# B&R Automation Studio project PLC code - cp (part 11)

#### InksCtrl.var
```iecst
VAR
	uiPosTachoCounterPrev : UINT;
	uiNegTachoCounterPrev : UINT;
	uiMode1Cycles : UINT;
	uiMode3Cycles : UINT;
	uiMode4Cycles : UINT;
	uiMode5Cycles : UINT;
	uiMode6Cycles : UINT;
	uiMode9Cycles : UINT;
	uiMode10Cycles : UINT;
	uiMode13Cycles : UINT;
	TON_AlrVacuum1 : TON;
	tonInkLevelBelowMinimum : TON;
	tonInkLevelBelowCloseMinimum : TON;
	TON_StabSolPid2Pos : TON; (*Vars Pressure Control*)
	TON_ChangeSPstarting : TON; (*It is a delay to recovery original set point after differential pressures*)
	TON_CloseSole : TON;
	tonInkLevelBelowMaximum : TON;
	TON_AlrTempGauge : TON;
	TON_HeaterStarts : TON;
	TON_AlrVacuum2 : TON;
	TON_OnReverseCappedCycle : TON; (*timer 30 min. It is cylce of reverse cleaning in Idle*)
	tonInkLevelAboveMaximum : TON;
	TON_DelayVacuum2Gauge : TON;
	tonInkLevelAboveMinimum : TON;
	TON_Stab2 : TON;
	TON_Stab1 : TON;
	TON_StabSolPid2Neg : TON;
	TON_TimeAfterCloseReliefValve : TON;
	TON_ChangeSPInDelta : TON; (*It is a delay to recovery original set point after differential pressures*) (*stChangeSPstarted : TON; *) (*It is a delay to recovery original set point after differential pressures*)
	TON_DelayVacuum1Gauge : TON;
	TON_ExecutionDelay : TON; (*Delay to activate the PID's in order to be sure to have proper configuration*)
	TON_AlrVacuumDiff2 : TON;
	TON_StabPsuOk : TON;
	TON_AlrNegDiff : TON;
	TON_StabSolPid1Neg : TON;
	TON_ChangeReverse : TON;
	TON_AlrDCDiff : TON;
	TON_AlrCriticalMeniscus2 : TON;
	TON_AlrNotDifTemp : TON;
	TON_TimeAlrDCStarting : TON;
	TON_AlrPosDiff : TON;
	TON_AlrIncoherTempHeat : TON;
	TON_AlrDifTemp : TON;
	TON_AlrVacuumDiff : TON;
	TON_StabSolPid1Pos : TON;
	TON_ChangeFillingControl : TON;
	TON_Reset : TON;
	TON_OnStateReverseFlow : TON; (*More time than 30 secs because It is coming back on reverse state *)
	TON_OnReverseCappedFinished : TON; (*timer 60 secs. It is time reverse cleaning in Idle*)
	TON_TimeExecutingReverseMan : TON;
	TON_Stopped : TON;
	TON_PressureReservoirStable : TON;
	TOF_IgnoreAlarmsCleaning : TOF;
	tonDrip : TON;
	parBar : REFERENCE TO stInksBarParams;
	inks : REFERENCE TO stInks;
	r_start_inks : R_TRIG;
	rSlopePumpNeg : REAL;
	rSPfillingPump : REAL; (*Value directly from Sw*)
	rPressureCollectorPos1 : REAL; (*REVISAR, sale un mensaje al traducir*)
	rSlopePumpPos : REAL;
	rSpeedNegCalc : REAL;
	rPressureCollectorPos2 : REAL; (*REVISAR, sale un mensaje al traducir*)
	rPressurePos : REAL;
	rPressureMen : REAL;
	rSP_NegPrimStabilizing : REAL;
	rSP_PosPrimStabilizing : REAL;
	rTankLevelmm : REAL;
	rSetPointFillingPump : REAL; (*Vars Temp Control*)
	rOrderBNegative : REAL;
	rVoltagePosPump : REAL;
	rOrderBPositiveStart : REAL;
	rOrderBPositive : REAL;
	rSP_Meniscus_PID : REAL;
	rMeniscusSp : REAL; (*Value directly from Sw*)
	rMeniscusPV : REAL;
	rVacuum2B : REAL;
	rSPTempTank : REAL;
	rHighPumpLimitNeg : REAL;
	rHighPumpLimitPos : REAL;
	rVoltageNegPump : REAL;
	rInputFilterVacuum2 : REAL;
	rLowPumpLimitNeg : REAL;
	parPidPos : REAL;
	parPidPosCopy : REAL;
	rInputFilterVacuum1 : REAL;
	parPidMeniscus : REAL;
	parPidMeniscusCopy : REAL;
	rSpeedPosCalc : REAL;
	parPidTemp : REAL;
	parPidTempCopy : REAL;
	rSPtemp : REAL; (*Temperature SetPoint*)
	rDutyCyclePreTune : REAL;
	rDutyCycleTempAux : REAL;
	rTankLevelPercent : REAL;
	rMeniscusError : REAL; (*Difference between Meniscus SetPint and PresentValue*)
	rLowPumpLimitPos : REAL;
	rSP_PressurePos_PID : REAL;
	rVacuum1B : REAL;
	pidParTempTank : MTPIDParametersType;
	pidParTemp : MTPIDParametersType;
	pidParMeniscus : MTPIDParametersType;
	pidParPresPos : MTPIDParametersType;
	fbFilterSpeedNeg : MTFilterMovingAverage;
	fbFilterMovingPressure2 : MTFilterMovingAverage;
	fbFilterMovingPressure1 : MTFilterMovingAverage;
	fbFilterLevelSensor : MTFilterMovingAverage;
	fbFilterSpeedPos : MTFilterMovingAverage;
	fbTempTunning : MTBasicsStepTuning;
	fb_PWM_Temp_Tank : MTBasicsPWM;
	fb_PWM_Temp : MTBasicsPWM;
	fb_PID_PresFilling : MTBasicsPID;
	fb_PID_Temp : MTBasicsPID;
	fb_PID_Tank_Temp : MTBasicsPID;
	fb_PID_Pres : MTBasicsPID;
	iTimeStopping : INT;
	tiTimePreviousExec : TIME;
	iTimesExecuted : INT;
	iBarNumberInBlock : INT;
	iCloseSoleW : INT;
	iDiffPulseTachoPos : INT;
	iDiffPulseTachoNeg : INT;
	iQuantityUpdatePidMeniscus : INT;
	iMs : UINT;
	tiDripTime : TIME;
	iSamplesVacuum2 : INT := 60;
	iQuantityUpdatePidPos : INT;
	iQuantityUpdatePidTemp : INT;
	iDisablePidW : INT;
	iStabSoleW : INT;
	tiDripTimeMax : TIME;
	iSamplesVacuum1 : INT := 1;
	iInkPreviousState : inksStateModes := INKS_STOPPED;
	xAuxSolenoidReverse : BOOL;
	xPossibleStart : BOOL;
	t_reset : BOOL;
	xEnableNegPID : BOOL;
	xPidTempTunning : BOOL;
	xAlarmEmptyTank : BOOL;
	xIgnoreAlarmsInCleaning : BOOL;
	xIAmInReverse : BOOL;
	xGoToStarted : BOOL; (*Meniscus is stable enough to go from Starting to Started*)
	xAnalogTankEmpty : BOOL;
	xEnablePwmTemp : BOOL;
	xAuxSolenoidDirect : BOOL;
	xHoldPos : BOOL; (*holding the PID in the reverse flows*)
	xAlarmFillTank : BOOL;
	xDrippingOrder : BOOL;
	xHoldMeniscus : BOOL;
	xPrimingStabilized : BOOL;
	xOutOfCriticalRange : BOOL;
	AuxiliarSolenoid : BOOL;
	xModesAlrDC : BOOL;
	xEnablePosPID : BOOL;
	xPressureReservoirStable : BOOL;
	xUpdatePidTemp : BOOL;
	mode1 : BOOL; (*INKS_STOPPED*)
	mode3 : BOOL; (*INKS_STARTING*)
	mode4 : BOOL; (*INKS_STARTED*)
	mode5 : BOOL; (*INKS_MANUAL_REVERSEFLOW*)
	mode6 : BOOL; (*INKS_AUTO_REVERSEFLOW*)
	mode9 : BOOL; (*INKS_STOPPING*)
	mode10 : BOOL; (*INKS_RUNNING_MANUAL*)
	mode13 : BOOL; (*INKS_PRIMING*)
	xStartHeating : BOOL; (*StartTemperature??*)
	xUpdatePidPos : BOOL;
	xStartTempPwm : BOOL;
	xReservoirModeActivated : BOOL;
	xStartTankHeating : BOOL;
	xUpdatePidMeniscus : BOOL;
	blink1s : Blink;
	ars_1020 : AutoResetSound; (*ars_1020: Auto reset sound for AlrVacuum1*)
	ars_1021 : AutoResetSound; (*ars_1021: Auto reset sound for AlrVacuum2*)
	ars_1022 : AutoResetSound;
	ars_1023 : AutoResetSound;
	ars_1010 : AutoResetSound;
	ars_1003 : AutoResetSound;
	ars_1009 : AutoResetSound;
	ars_1019 : AutoResetSound; (*Auto resete alarm for refilling tank, it is activated when level is lower than max*)
	ars_1016 : AutoResetSound; (*ars_1017 : AutoResetSound;*)
	ars_1013 : AutoResetSound; (*ars_1014 : AutoResetSound;*)
	ars_1012 : AutoResetSound;
	ars_1011 : AutoResetSound;
	ars_1008 : AutoResetSound;
	ars_1015 : AutoResetSound;
	ars_1018 : AutoResetSound;
	ars_1007 : AutoResetSound;
	ars_1006 : AutoResetSound;
	ars_1005 : AutoResetSound;
	ars_1004 : AutoResetSound;
	ars_1001 : AutoResetSound;
	ars_1002 : AutoResetSound;
	ars_1000 : AutoResetSound;
	TON_AlrTempTankTempSensorError : TON;
	resetedAlarms : stInksAlarmsList;
	resetedAlarmsSummary : stEFI_AlarmSummary;
	resetedOut : stInksSignalsOut;
	resetedStatus : stInksStatus;
	stEventLogCritical : EventLog_typ;
	stStopAlarmsLog : EventLog_typ;
	stEventLog : EventLog_typ;
	stEventLogPos : EventLog_typ;
	stEventLogNeg : EventLog_typ;
	strAux : STRING[129];
	xUpdateSpPriming : BOOL;
	xStateReverseFlow : BOOL := FALSE;
	iReasonStop : UDINT;
	iReasonCritical : UDINT;
	iReasonWarning : UDINT;
	xReservoirParamsNeeded : BOOL;
	iReasonToSound : UDINT;
	tonAlrNotHeating : TON;
	TON_AlrDifTempTank : TON;
	TON_AlrDifTempTank2 : TON;
	TON_AlrTempTankMax : TON;
	ars_1017 : AutoResetSound;
	TON_AlrTempHeaterMax : TON;
	TON_AlrIncoherTempTank : TON;
	ars_1024 : AutoResetSound;
	ars_1025 : AutoResetSound;
	ars_1026 : AutoResetSound;
	ars_1027 : AutoResetSound;
	TON_OverPressureDelay : TON;
	TON_AlrDifTempExcessiv : TON;
	TON_AlrNotDifTempExcessiv : TON;
	rVacuumSensorMax : REAL;
	iReasonRunning : UINT;
	iReasonEnableNegPID : USINT;
	iReasonEnablePosPID : USINT;
	iReasonRunningAuto : USINT;
	xRunningAuto : BOOL;
	RTInfo_0 : RTInfo;
	rPeriode : REAL;
	iPeriode : UINT;
	TON_AlrHeaterOFF : TON;
	TON_AlrChillerPrintheadsOFF : TON;
	tonStabInkStartUp : TON; (*Timer to define stable enough to modify the set point*)
	tonNotStabInkStartUp : TON; (*Timer to define NOT stable enough to modify the set point*)
	tonUstabInkStartUp : TON; (*Inks unstable so long, so automatic startup is cancelled*)
	rMeniscusStartUpStep : REAL;
	xStabMeniscus : BOOL;
END_VAR
```

#### Inks.fun
```iecst
FUNCTION inkStateValue : INT (*TODO: Add your comment here*) (*$GROUP=User,$CAT=User,$GROUPICON=User.png,$CATICON=User.png*)
	VAR_INPUT
		inkState : inksStateModes;
	END_VAR
END_FUNCTION

FUNCTION stPIDParamId : REAL (*TODO: Add your comment here*) (*$GROUP=User,$CAT=User,$GROUPICON=User.png,$CATICON=User.png*)
	VAR_INPUT
		parPid : stPIDParam;
	END_VAR
END_FUNCTION

FUNCTION timeToStartPWM : BOOL (*TODO: Add your comment here*) (*$GROUP=User,$CAT=User,$GROUPICON=User.png,$CATICON=User.png*)
	VAR_INPUT
		iItemNumber : INT;
		iTotalItems : INT;
		iTaskCycle : UINT; (*Task cycle in ms*)
	END_VAR
	VAR_IN_OUT
		iMsInCycle : UINT;
	END_VAR
END_FUNCTION

FUNCTION stPIDParamToMTPIDParameters : BOOL (*Void function to fill the value of stPIDParam in a  MTPIDParametersType*)
	VAR_INPUT
		pidParam : REFERENCE TO stPIDParam;
		MTPIDparam : REFERENCE TO MTPIDParametersType;
	END_VAR
END_FUNCTION
```

#### alarmsSound.st
```iecst
ACTION alarmsSound:

	///Auto reset sound management. All alarms need to work with mute option
	ars_1000(xAlarm:=inks.Al.xAlrTankCloseToEmpty,		xSilence:=inks.commands.xMute);
	ars_1001(xAlarm:=inks.Al.xAlrTankEmpty,				xSilence:=inks.commands.xMute);
	ars_1002(xAlarm:=inks.Al.xAlrLevelSensorError,		xSilence:=inks.commands.xMute);
	ars_1003(xAlarm:=inks.Al.xAlrIncoherTempHeat,		xSilence:=inks.commands.xMute);
	ars_1004(xAlarm:=inks.Al.xAlrNoInkNoCleanManif,		xSilence:=inks.commands.xMute);
	ars_1005(xAlarm:=inks.Al.xAlrNoRecircStop,			xSilence:=inks.commands.xMute);
	ars_1006(xAlarm:=inks.Al.xAlrStopRecircNoInk,		xSilence:=inks.commands.xMute);
	ars_1007(xAlarm:=inks.Al.xAlrNoInkNoCleanManif,		xSilence:=inks.commands.xMute);
	ars_1008(xAlarm:=inks.Al.xAlrOverPressure,			xSilence:=inks.commands.xMute);
	//ars_1009(xAlarm:=,			xSilence:=);
	ars_1010(xAlarm:=inks.Al.xAlrVacuumSensor1,			xSilence:=inks.commands.xMute);
	ars_1011(xAlarm:=inks.Al.xAlrVacuumSensor2,			xSilence:=inks.commands.xMute);
	ars_1012(xAlarm:=inks.Al.xAlrTempSensor,			xSilence:=inks.commands.xMute);
	ars_1013(xAlarm:=inks.Al.xAlrPrintHeadPsuFailure,	xSilence:=inks.commands.xMute);
	//ars_1014(xAlarm:=inks.Al.xAlrNoRecirculation,		xSilence:=inks.commands.xMute);
	ars_1015(xAlarm:=inks.Al.xAlrPumpsDCError,			xSilence:=inks.commands.xMute);
	ars_1016(xAlarm:=inks.Al.xAlrBrokenMeniscus,		xSilence:=inks.commands.xMute);
	ars_1017(xAlarm:=inks.Al.xAlrHeaterTankReachsMaxTemp,xSilence:=inks.commands.xMute);
	ars_1018(xAlarm:=inks.Al.xAlrKlixonTriggered,		xSilence:=inks.commands.xMute);
	ars_1019(xAlarm:=inks.Al.xAlrTankToFillIn,			xSilence:=inks.commands.xMute);
	ars_1020(xAlarm:=inks.Al.xAlrVacuum1,				xSilence:=inks.commands.xMute);
	ars_1021(xAlarm:=inks.Al.xAlrVacuum2,				xSilence:=inks.commands.xMute);
	ars_1022(xAlarm:=inks.Al.xAlrTempTankSensor,		xSilence:=inks.commands.xMute);
	ars_1023(xAlarm:=inks.Al.xAlrHeaterReachsMaxTemp,	xSilence:=inks.commands.xMute);
	ars_1024(xAlarm:=inks.Al.xAlrIncoherTempTank,		xSilence:=inks.commands.xMute);
	ars_1025(xAlarm:=inks.Al.xAlrHeaterOutFault,		xSilence:=inks.commands.xMute);
	ars_1026(xAlarm:=inks.Al.xAlrDifCtrlTempExcessive,	xSilence:=inks.commands.xMute);
	ars_1027(xAlarm:=inks.Al.xAlrMaintenanceModeActive,	xSilence:=inks.commands.xMute);

	//The alarms to make sound due to the Inks
	iReasonToSound.0 := ars_1000.xAlarmSound;
	iReasonToSound.1 := ars_1001.xAlarmSound;
	iReasonToSound.2 := ars_1002.xAlarmSound;
	iReasonToSound.3 := ars_1003.xAlarmSound;
	iReasonToSound.4 := ars_1004.xAlarmSound;
	iReasonToSound.5 := ars_1005.xAlarmSound;
	iReasonToSound.6 := ars_1006.xAlarmSound;
	iReasonToSound.7 := ars_1007.xAlarmSound;
	iReasonToSound.8 := ars_1008.xAlarmSound;
	iReasonToSound.9 := ars_1009.xAlarmSound;
	iReasonToSound.10 := ars_1010.xAlarmSound;
	iReasonToSound.11 := ars_1011.xAlarmSound;
	iReasonToSound.12 := ars_1012.xAlarmSound;
	iReasonToSound.13 := ars_1013.xAlarmSound;
	//iReasonToSound.14 := ars_1014.xAlarmSound;
	iReasonToSound.15 := ars_1015.xAlarmSound;
	iReasonToSound.16 := ars_1016.xAlarmSound;
	iReasonToSound.17 := ars_1017.xAlarmSound;
	iReasonToSound.18 := ars_1018.xAlarmSound;
	iReasonToSound.19 := ars_1019.xAlarmSound;
	iReasonToSound.20 := ars_1020.xAlarmSound;
	iReasonToSound.21 := ars_1021.xAlarmSound;
	iReasonToSound.22 := ars_1022.xAlarmSound;
	iReasonToSound.23 := ars_1023.xAlarmSound;
	iReasonToSound.24 := ars_1024.xAlarmSound;
	iReasonToSound.25 := ars_1025.xAlarmSound;
	iReasonToSound.26 := ars_1026.xAlarmSound;
	iReasonToSound.27 := ars_1027.xAlarmSound;

	inks.AlSummary.xAlarmSound:=iReasonToSound > 0;

END_ACTION
```

#### alarmsSummary.st
```iecst
ACTION alarmsSummary:

	//FILL AlarmSummary data

	//Inks critical alarm used to stop the ink sistem
	iReasonCritical.0 := inks.Al.xAlrTankEmpty;
	iReasonCritical.1 := inks.Al.xAlrStopRecircNoInk;
	iReasonCritical.2 := inks.Al.xAlrIncoherTempHeat;
	iReasonCritical.3 := inks.Al.xAlrVacuum1;
	iReasonCritical.4 := inks.Al.xAlrVacuum2;
	iReasonCritical.5 := inks.Al.xAlrVacuumSensor1;
	iReasonCritical.6 := inks.Al.xAlrVacuumSensor2;
	iReasonCritical.7 := inks.Al.xAlrTempSensor;
	iReasonCritical.8 := inks.Al.xAlrBrokenMeniscus;
	iReasonCritical.9 := inks.Al.xAlrOverPressure;
	iReasonCritical.10 := inks.Al.xAlrLevelSensorError;
	iReasonCritical.11 := inks.Al.xAlrTankDigitalSensorsError;
	iReasonCritical.12 := inks.Al.xAlrPumpsDCError;
	iReasonCritical.13 := FALSE;
	iReasonCritical.14 := FALSE;

	inks.AlSummary.xAlarmCritical :=  iReasonCritical > 0;
	//Register the reason of the Critical Alarm
	IF inks.status.iInkState <> INKS_STOPPED  AND EDGEPOS(inks.AlSummary.xAlarmCritical) THEN
		inks.AlSummary.iReasonCritical := iReasonCritical;
		LogCriticalAlarm;
	ELSIF EDGEPOS(inks.status.iInkState = INKS_STARTED AND NOT inks.AlSummary.xAlarmCritical) THEN
		inks.AlSummary.iReasonCritical := 0;
	END_IF

	iReasonWarning.0 := inks.Al.xAlrTankToFillIn;
	iReasonWarning.1 := inks.Al.xAlrDiffInCtrlTempTank;
	iReasonWarning.2 := inks.Al.xAlrDiffInCtrlTemp;
	iReasonWarning.3 := inks.Al.xAlrNoInkNoCleanManif;
	iReasonWarning.4 := inks.Al.xAlrKlixonTriggered;
	iReasonWarning.5 := inks.Al.xAlrTempTankSensor;
	iReasonWarning.6 := inks.Al.xAlrNoRecirculation;
	iReasonWarning.7 := inks.Al.xAlrHeaterReachsMaxTemp;
	iReasonWarning.8 := inks.Al.xAlrIncoherTempTank;
	iReasonWarning.9 := inks.Al.xAlrHeaterTankReachsMaxTemp;
	iReasonWarning.10 := inks.Al.xAlrMaintenanceModeActive;
	iReasonWarning.11 := inks.Al.xHeaterOff; // NOZOMITWO-1410
	iReasonWarning.12 := inks.Al.xAlrDiffVacuum;

	//Warning alarms (used in sound alarms).
	inks.AlSummary.xAnyWarning:= iReasonWarning > 0;

	// Ink Stop Alarms are used to stop of printing state
	iReasonStop.0 := iReasonCritical > 0;
	iReasonStop.1 := inks.Al.xAlrHeaterOutFault;
	iReasonStop.2 := inks.Al.xAlrPrintHeadPsuFailure;
	iReasonStop.3 := inks.Al.xAlrDifCtrlTempExcessive;
	iReasonStop.4 := EDGENEG(inks.ordersSw.xStartInks) AND NOT (iReasonCritical > 0);
	iReasonStop.5 := inks.parSw.Config.iInkType = 0;
	iReasonStop.6 := inks.parSw.Config.iPrintHeadType = 0;
	iReasonStop.7 := inks.Al.xAlrNoRecircStop;
	iReasonStop.8 := inks.Al.xAlrTankCloseToEmpty;
	iReasonStop.9 := inks.Al.xAlrPrintHeadsChillerStopped;

	IF iReasonStop > 0 AND inks.status.xEnabledBarToPrint THEN
		inks.AlSummary.xAlarmStop:= TRUE;
	ELSIF inks.commands.xErrorRst THEN
		inks.AlSummary.xAlarmStop:= FALSE;
	END_IF

	//Register the reason of the Stop Alarm
	IF inks.status.iInkState <> INKS_STOPPED  AND EDGEPOS(inks.AlSummary.xAlarmStop) THEN
		//Register the reason of the Stop Alarm
		LogStopAlarm;
		inks.AlSummary.iReasonStop[0] := iReasonStop;
	ELSIF EDGEPOS(inks.status.iInkState = INKS_STARTING AND NOT inks.AlSummary.xAlarmStop) THEN
		inks.AlSummary.iReasonStop[0] := 0;
	END_IF

	inks.AlSummary.xAnyAlarm:= inks.AlSummary.xAlarmCritical OR inks.AlSummary.xAlarmStop OR inks.AlSummary.xAnyWarning;

END_ACTION
```

#### calculations.st
```iecst
ACTION calculations:

	IF NOT xIAmInReverse THEN
		rPressureCollectorPos1:= rVacuum1B ;
		rPressureCollectorPos2:= rVacuum2B;
	ELSE
		rPressureCollectorPos1:= rVacuum2B;
		rPressureCollectorPos2:= rVacuum1B;
	END_IF
	inks.status.rMeniscus:= (-1)*((rPressureCollectorPos1 + rPressureCollectorPos2)/2);

	inks.status.rDeltaPressure:= ABS (rPressureCollectorPos1 - rPressureCollectorPos2);
	rSPfillingPump:=inks.parSw.PosPump.rSetPoint;

	rMeniscusPV:=			inks.status.rMeniscus;

	//DELOREAN-1961
	IF NOT inks.parSw.xActMaintenanceMode THEN
		rSPtemp:= inks.parSw.Temp.rSetPointTemp;
	ELSE
		rSPtemp:= inks.parSw.Temp.rSetPointTempMaintenance;
	END_IF

	// Ink Heater Tank works at the same set point than Ink Heater Bar. For this reason, they use same values from GUI
	rSPTempTank:=			inks.parSw.Temp.rSetPointTemp;
	rMeniscusError:=		ABS(rMeniscusSp - rMeniscusPV);

	//Call the tachometer calculation of the pump
	tachoCalculations;

END_ACTION

ACTION tachoCalculations:
	IF NOT inks.parameters.xEnabledTachoSignals THEN
		RETURN;
	END_IF

	// Speedometer  Speedometer  Speedometer  Speedometer  Speedometer  Speedometer  Speedometer Speedometer  Speedometer  Speedometer Speedometer Speedometer  Speedometer
	//
	//Change units from pulses per rev to rpm (The digital counter is configured as event counter so if the ink pump has 2 PULSES per rev, is measuring 4 EVENTS per rev)
	iDiffPulseTachoNeg:= SAFE_UINTDIFF(uiLastValue:= inks.signals.in.iTachNegative, uiPrevValue:= uiNegTachoCounterPrev);
	rSpeedNegCalc:= UINT_TO_REAL(iDiffPulseTachoNeg) * 1000 * 60 / TIME_TO_REAL(clock_ms() - tiTimePreviousExec) / 4;

	iDiffPulseTachoPos:= SAFE_UINTDIFF(uiLastValue:= inks.signals.in.iTachFilling, uiPrevValue:= uiPosTachoCounterPrev);
	rSpeedPosCalc:= UINT_TO_REAL(iDiffPulseTachoPos) * 1000 * 60 / TIME_TO_REAL(clock_ms() - tiTimePreviousExec) / 4;

	//Filters to remove tach signal sensibility
	fbFilterSpeedNeg(Enable:=TRUE,
		In:=rSpeedNegCalc,
		WindowLength:=30 , //20*48:=1second
		);
	inks.status.NegPump.rSpeedNeg := fbFilterSpeedNeg.Out;

	fbFilterSpeedPos(Enable:=TRUE ,
		In:=rSpeedPosCalc,
		WindowLength:=30 , //20*48:=1second
		);
	inks.status.PosPump.rSpeedPos := fbFilterSpeedPos.Out;

	uiNegTachoCounterPrev := inks.signals.in.iTachNegative;
	uiPosTachoCounterPrev := inks.signals.in.iTachFilling;
	tiTimePreviousExec := clock_ms();

END_ACTION
```

#### controlMode.st
```iecst
ACTION controlMode:

	inks.status.iInkState := LIMIT(1,inks.status.iInkState,13);

	//Just change ReservoirMode when stopped
	IF inks.status.iInkState = INKS_STOPPED THEN
		xReservoirModeActivated:= inks.parameters.xReservoirMode;
	END_IF

	//Control of the different working methods of the ink system:
	inks.status.xEnabledBarToPrint := inks.parSw.xEnabledBarToPrint;
	inks.status.xColorLoadedInJob := inks.parSw.xColorLoadedInJob;
	inks.status.xActTestMode := inks.parSw.xActTestMode;
	inks.status.xActMaintenanceMode := inks.parSw.xActMaintenanceMode;

	//MODE 9: STOPPING THE SYSTEM. The mode is used before the system is stopped.
	IF xRunningAuto AND (NOT inks.ordersSw.xStartInks OR inks.AlSummary.xAlarmCritical) THEN
		iInkPreviousState := inks.status.iInkState;
		inks.status.iInkState := INKS_STOPPING;
	END_IF

	//MODE1: SYSTEM STOPPED
	//Stop in cleaning minifolds and canlcel order or OverPresure alarm appear
	IF 	((NOT inks.ordersSw.xStartManual OR inks.Al.xAlrOverPressure) AND inks.status.iInkState = INKS_RUNNING_MANUAL) THEN //Stop in any others ink state if any crital alarm appear
		iInkPreviousState := inks.status.iInkState;
		inks.status.iInkState := INKS_STOPPED;
		removeOrders;
	END_IF

	TON_Stopped.IN:= inks.status.iInkState = INKS_STOPPING;
	TON_Stopped.PT:= INT_TO_TIME(inks.parameters.iTimeStopping);
	TON_Stopped();

	iTimeStopping:=TIME_TO_INT(TON_Stopped.ET);
	IF TON_Stopped.Q THEN
		iInkPreviousState := inks.status.iInkState;
		inks.status.iInkState := INKS_STOPPED ;
	END_IF

	//MODE3 AND MODE13: INK SYSTEM START. When the system is charged we can start it.
	xPossibleStart:=  inks.status.iInkState = INKS_STOPPED AND
					(inks.status.Tank.xMinLevel OR inks.status.xActTestMode) AND
					NOT inks.Al.xAlrOverPressure;

	r_start_inks(CLK:= inks.ordersSw.xStartInks);

	IF xPossibleStart AND r_start_inks.Q THEN
		//Depending on the type of the system, go to priming or not
		IF inks.parameters.Priming.xSystemNeedsPriming THEN
			inks.status.iInkState := INKS_PRIMING;
		ELSE
			inks.status.iInkState := INKS_STARTING;
		END_IF
		iInkPreviousState := inks.status.iInkState;
	END_IF

	//Go to Starting from the Priming state
	IF inks.status.iInkState = INKS_PRIMING AND (inks.status.rMeniscus<-10) THEN
		inks.status.iInkState := INKS_STARTING;
	END_IF

	//If the system is not ready to start, fall down the start command
	IF (r_start_inks.Q AND inks.status.iInkState <> INKS_STARTING) OR inks.status.iInkState=INKS_STOPPED THEN
		inks.ordersSw.xStartInks:=FALSE;
	END_IF

	//MODE4: When the system is stabilized we are in the mode4.
	IF 	(inks.status.iInkState = INKS_STARTING AND (xGoToStarted OR xPrimingStabilized) ) OR
		(inks.status.iInkState = INKS_MANUAL_REVERSEFLOW AND EDGENEG(inks.ordersSw.xOrderReverseMan) ) OR
		(inks.status.iInkState = INKS_AUTO_REVERSEFLOW AND NOT inks.commands.xOrderCleaning) OR
		(inks.status.iInkState = INKS_AUTO_REVERSEFLOW AND NOT inks.status.Reverse.xStartOnReverseCapped) THEN

			iInkPreviousState := inks.status.iInkState;
			inks.status.iInkState := INKS_STARTED;
	END_IF

	//MODE 5: MANUAL REVERSE FLOW. When the interface button is pressed, we change the flow direction.
	IF inks.status.iInkState = INKS_STARTED AND EDGEPOS(inks.ordersSw.xOrderReverseMan) THEN
		xPressureReservoirStable:=FALSE;
		iInkPreviousState := inks.status.iInkState;
		inks.status.iInkState := INKS_MANUAL_REVERSEFLOW;
	END_IF

	//MODE 6: AUTOMATIC REVERSE FLOW. Is done on printheads cleaning.
	IF inks.commands.xOrderCleaning AND inks.parSw.xOnReverseCleaning THEN
		inks.status.Reverse.xOnReverseCleaning:=TRUE;
	ELSIF inks.parSw.xOnReverseCapped AND inks.parameters.xBlockInCap THEN
		inks.status.Reverse.xOnReverseCapped:= TRUE;
	ELSE
		inks.status.Reverse.xOnReverseCleaning:=FALSE;
		inks.status.Reverse.xOnReverseCapped:=FALSE;
	END_IF

	//Reverse flow just works when ink is started
	IF inks.status.iInkState = INKS_STARTED AND ( inks.status.Reverse.xOnReverseCleaning OR (inks.status.Reverse.xOnReverseCapped AND  inks.status.Reverse.xStartOnReverseCapped ) ) THEN
		xPressureReservoirStable:=FALSE;
		iInkPreviousState := inks.status.iInkState;
		inks.status.iInkState := INKS_AUTO_REVERSEFLOW ;
	END_IF

	//MODE 10: Running Manual
	IF 	inks.status.iInkState = INKS_STOPPED AND (inks.status.Tank.xMinLevel OR  inks.status.xActTestMode) AND
		inks.ordersSw.xStartManual  THEN
			iInkPreviousState := inks.status.iInkState;
			inks.status.iInkState := INKS_RUNNING_MANUAL;
	END_IF

	// Solenid direction management
	//
	IF (inks.status.iInkState = INKS_STOPPED AND inks.status.xInksRunning) OR inks.status.iInkState = INKS_STOPPING  THEN
		inks.status.iDirection := INKSDIR_STOP;
	END_IF

	//When ink flow is direct xInksManifoldsCleaningInReverse is false and everytime that is stopped is restored to false
	//just in case of pareameter, ink flow is reverted or not for cleaning manifolds
	// Pending to update parameter to iInksManifoldsCleaningReverted;
	inks.status.Reverse.xReverseOnManual:= inks.parSw.xReverseOnManual;

	IF 	inks.status.iInkState = INKS_PRIMING OR
		inks.status.iInkState = INKS_STARTING OR
		inks.status.iInkState = INKS_STARTED OR
		(inks.status.iInkState = INKS_RUNNING_MANUAL AND NOT inks.status.Reverse.xReverseOnManual ) THEN
		inks.status.iDirection := INKSDIR_DIRECT;
	END_IF

	IF (inks.status.iInkState = INKS_MANUAL_REVERSEFLOW OR inks.status.iInkState = INKS_AUTO_REVERSEFLOW) OR
		(inks.status.iInkState = INKS_RUNNING_MANUAL AND inks.status.Reverse.xReverseOnManual ) THEN
		inks.status.iDirection := INKSDIR_REVERSE;
	END_IF

	//Defining the system is running in auto mode
	iReasonRunningAuto.0 := inks.status.iInkState = INKS_STARTING;
	iReasonRunningAuto.1 := inks.status.iInkState = INKS_PRIMING;
	iReasonRunningAuto.2 := inks.status.iInkState = INKS_STARTED;
	iReasonRunningAuto.3 := inks.status.iInkState = INKS_MANUAL_REVERSEFLOW;
	iReasonRunningAuto.4 := inks.status.iInkState = INKS_AUTO_REVERSEFLOW;
	xRunningAuto := iReasonRunningAuto > 0;

	//Conditions to start de ink system
	iReasonRunning.0 := inks.status.iInkState = INKS_STOPPING;
	iReasonRunning.1 := inks.status.iInkState = INKS_RUNNING_MANUAL;
	inks.status.xInksRunning := xRunningAuto OR iReasonRunning > 0;

	// If running in auto, remove order to run manual
	IF xRunningAuto THEN
		inks.ordersSw.xStartManual := FALSE;
	END_IF

	xStateReverseFlow:= inks.status.iInkState = INKS_MANUAL_REVERSEFLOW OR inks.status.iInkState = INKS_AUTO_REVERSEFLOW;

	//manual reverse time management
	IF inks.status.iInkState = INKS_STOPPED THEN
		inks.status.Reverse.xReverseManFinished := TRUE;
	ELSIF inks.ordersSw.xOrderReverseMan THEN
		inks.status.Reverse.xReverseManFinished := FALSE;
	END_IF

	inks.status.Reverse.xReverseMan := (inks.status.iInkState = INKS_MANUAL_REVERSEFLOW);

	TON_TimeExecutingReverseMan.IN:= inks.status.iInkState = INKS_MANUAL_REVERSEFLOW;
	TON_TimeExecutingReverseMan.PT:= MAX(inks.parSw.tiReverseManual, T#3s);
	TON_TimeExecutingReverseMan();
	inks.status.tiInReverseManual:=TON_TimeExecutingReverseMan.ET;
	IF TON_TimeExecutingReverseMan.Q THEN
		// It sets inks.commnads.xOrderReverseMan FALSE because is a latched
		inks.ordersSw.xOrderReverseMan:=FALSE;
		inks.status.Reverse.xReverseManFinished := TRUE;
	END_IF

	//Unestable ink system state.
	inks.status.xUnstableInkState := (inks.Al.xAlrDiffVacuum OR inks.Al.xAlrDiffInCtrlTemp) AND inks.status.xInksRunning;

	//Update values for the current control cycle
	//We match the different values of the variable iInkstate with internal variables
	mode1 := inks.status.iInkState = INKS_STOPPED;
	mode3 := inks.status.iInkState = INKS_STARTING;
	mode4 := inks.status.iInkState = INKS_STARTED;
	mode5 := inks.status.iInkState = INKS_MANUAL_REVERSEFLOW;
	mode6 := inks.status.iInkState = INKS_AUTO_REVERSEFLOW;
	mode9 := inks.status.iInkState = INKS_STOPPING;
	mode10:= inks.status.iInkState = INKS_RUNNING_MANUAL;
	mode13:= inks.status.iInkState = INKS_PRIMING;

	//The vacuuum sensor readings are changed if we are in reverse flow.
	TON_ChangeReverse(IN:=mode5 OR mode6, PT:= T#100MS);
	xIAmInReverse:=TON_ChangeReverse.Q;

	// xOrderDrip when is cleaning while 50 secs, from start dropping to suction finished
	TOF_IgnoreAlarmsCleaning(IN:= inks.commands.xOrderDrip, PT:= T#50s);
	xIgnoreAlarmsInCleaning:=TOF_IgnoreAlarmsCleaning.Q;

	// When GUI sends Idle reverse function, It sets xOnReverseCapped and then is updated GUI
	// and started reverse flow OF 60 secs every 30 MIN
	//
	IF inks.parSw.xOnReverseCapped AND NOT TON_OnReverseCappedFinished.Q THEN
		inks.status.Reverse.xStartOnReverseCappedCycle:=TRUE;
	ELSE
		inks.status.Reverse.xOnReverseCapped:=FALSE;
		inks.status.Reverse.xStartOnReverseCapped:=FALSE;
		inks.status.Reverse.xStartOnReverseCappedCycle:=FALSE;
	END_IF
	// timer of cycles
	TON_OnReverseCappedCycle(IN:=inks.status.Reverse.xStartOnReverseCappedCycle, PT:=T#30M);

	IF TON_OnReverseCappedCycle.Q AND
	    NOT xDrippingOrder AND
		(NOT inks.ordersSw.xStartManual) AND
		(NOT inks.ordersSw.xOrderReverseMan) THEN

		inks.status.Reverse.xStartOnReverseCapped:=TRUE;
		inks.status.Reverse.xOnReverseCapped:=TRUE;

	END_IF
	// reverse flow timer management in cap position. Idle reverse function in GUI
	TON_OnReverseCappedFinished(IN:=inks.status.Reverse.xStartOnReverseCapped, PT:=T#60S);
	IF TON_OnReverseCappedFinished.Q THEN
		//It stops reverse flow and initialize inputs timers
		inks.status.Reverse.xOnReverseCapped:=FALSE;
		inks.status.Reverse.xStartOnReverseCapped:=FALSE;
		inks.status.Reverse.xStartOnReverseCappedCycle:=FALSE;
		inks.status.Reverse.xOnReverseAuto:=TRUE;
	END_IF

	TON_OnStateReverseFlow(IN:=inks.status.Reverse.xOnReverseAuto);

	IF TON_OnStateReverseFlow.Q THEN
		inks.status.Reverse.xOnReverseAuto:=FALSE;
	END_IF
	inks.status.iInkStateSw := inkStateValue(inks.status.iInkState);

	IF inks.parameters.xDebugMode THEN RETURN; END_IF

	//Information just if debugging
	IF mode1 THEN 	uiMode1Cycles:=uiMode1Cycles+1; END_IF
	IF mode3 THEN 	uiMode3Cycles:=uiMode3Cycles+1; END_IF
	IF mode4 THEN 	uiMode4Cycles:=uiMode4Cycles+1; END_IF
	IF mode5 THEN 	uiMode5Cycles:=uiMode5Cycles+1; END_IF
	IF mode6 THEN 	uiMode6Cycles:=uiMode6Cycles+1; END_IF
	IF mode9 THEN 	uiMode9Cycles:=uiMode9Cycles+1; END_IF
	IF mode10 THEN 	uiMode10Cycles:=uiMode10Cycles+1; END_IF
	IF mode13 THEN 	uiMode13Cycles:=uiMode13Cycles+1; END_IF

END_ACTION

ACTION removeOrders:
	inks.ordersSw.xStartManual :=	FALSE;
	inks.ordersSw.xOrderReverseMan := 			FALSE;
END_ACTION
```

#### dripControl.st
```iecst
ACTION dripControl:

	//  The bar waits an OrderDrip while any of the bars in the same block has to drip.
	// Each bar delays the start of the dripping taking into account its dripping time and the MaxDripTime
	// The Block is the responsible of removing the OrderDrip with a timer of the MaxDripTime of its bars

	// Just in case of Drip time is upper to 0 then It sends drip order to pressure control. Jira 784
	tonDrip.IN := inks.status.xInksRunning AND inks.commands.xOrderDrip AND TON_TimeAfterCloseReliefValve.Q AND (inks.status.tiDriptime>0);
	tonDrip.PT := tiDripTimeMax - tiDripTime; //Using the internal vars. Cheched the limits in ConversionsPre
	tonDrip();
	xDrippingOrder := tonDrip.Q;

	inks.status.xDripping := xDrippingOrder;

END_ACTION
```

#### inkLevel.st
```iecst
ACTION inkLevel:

	IF tonInkLevelAboveMinimum.Q THEN
		inks.status.Tank.xMinLevel := TRUE;
	END_IF
	IF tonInkLevelBelowMinimum.Q THEN
		inks.status.Tank.xMinLevel := FALSE;
	END_IF

	IF tonInkLevelAboveMinimum.Q THEN
		inks.status.Tank.xCloseToMinLevel := TRUE;
	END_IF
	IF tonInkLevelBelowCloseMinimum.Q THEN
		inks.status.Tank.xCloseToMinLevel := FALSE;
	END_IF

	IF tonInkLevelAboveMaximum.Q THEN
		inks.status.Tank.xMaxLevel := TRUE;
	END_IF
	IF tonInkLevelBelowMaximum.Q THEN
		inks.status.Tank.xMaxLevel := FALSE;
	END_IF

	//0=Empty ; 1=Min; 2=Full; 3=Non valid level
	IF parBar.xTypeTankSensorDigital THEN

		tonInkLevelAboveMaximum(IN:= inks.signals.in.xMaxLevel, PT:=T#35s);
		tonInkLevelBelowMaximum(IN:= NOT inks.signals.in.xMaxLevel, PT:=T#1m);

		tonInkLevelBelowCloseMinimum(IN:= NOT inks.signals.in.xMinLevel, PT:=T#10s);

		tonInkLevelAboveMinimum(IN:= inks.signals.in.xMinLevel, PT:=T#35s);
		tonInkLevelBelowMinimum(IN:= NOT inks.signals.in.xMinLevel, PT:=T#1m);

		IF NOT inks.status.Tank.xMinLevel AND NOT inks.status.Tank.xMaxLevel THEN inks.status.Tank.iStatusTankDigital := 0; END_IF
		IF inks.status.Tank.xMinLevel AND NOT inks.status.Tank.xMaxLevel THEN 	inks.status.Tank.iStatusTankDigital := 1; END_IF
		IF inks.status.Tank.xMinLevel AND inks.status.Tank.xMaxLevel THEN 		inks.status.Tank.iStatusTankDigital := 2; END_IF
		IF NOT inks.status.Tank.xMinLevel AND inks.status.Tank.xMaxLevel THEN 	inks.status.Tank.iStatusTankDigital := 3; END_IF

	ELSE
		inks.status.Tank.iStatusTankDigital := 3;

		tonInkLevelAboveMaximum(IN:= inks.status.Tank.iDipositLevel>42, PT:=T#10s);
		tonInkLevelBelowMaximum(IN:= inks.status.Tank.iDipositLevel<40, PT:=T#10s);

		// Ink level can have 1% of change by bars movement, so 7% with 4% is more robust
		tonInkLevelBelowCloseMinimum(IN:= inks.status.Tank.iDipositLevel<=7, PT:=T#10s);

		tonInkLevelAboveMinimum(IN:= inks.status.Tank.iDipositLevel>9, PT:=T#10s);
		tonInkLevelBelowMinimum(IN:= inks.status.Tank.iDipositLevel<4, PT:=T#10s);
	END_IF

	//NOTE: When implement xTypeTankSensorAnalog, reset xMinLevel and xMaxLevel from Digital

END_ACTION
```

#### Main.st
```iecst
PROGRAM _INIT
	RTInfo_0(enable :=TRUE );
	rPeriode:= UDINT_TO_REAL (RTInfo_0.cycle_time)/1000;  // Cycle time in microseconds
	iPeriode := REAL_TO_UINT(rPeriode);
END_PROGRAM

PROGRAM _CYCLIC

	//Reference working data to the general data
	inks ACCESS ADR(gInks[gIndexInks]);
	parBar ACCESS ADR(inks.parameters.parBar);

	inks.status.xBarInstalled:=inks.parSw.Config.iMappingBar >= 1 AND inks.parSw.Config.iMappingBar <= MAX_LAST_INK ;

	//IMPORTANT: In printHeadData MUST be referenced the parBar (in Permanent Variable)
	IF NOT inks.status.xBarInstalled THEN
		inks.Al:=resetedAlarms;
		inks.AlSummary:=resetedAlarmsSummary;
		inks.status:=resetedStatus;
		inks.signals.out:=resetedOut;
		gIndexInks := gIndexInks + 1; //Point to the next Bar
		RETURN;
	END_IF

	//Reset all alarms if error reset received
	IF inks.commands.xErrorRst THEN
		inks.Al:=resetedAlarms;
	END_IF

	safetyPre;

	inkLevel;
	controlMode;
	conversionsPre;
	calculations;
	dripControl;

	startUp;

	reservoirMode;

	pressureControl;
	tempControl;
	solenoids;

	conversionsPost;
	powPrintHeads;
	alarms;
	alarmsSummary;
	alarmsSound;

	iTimesExecuted:=iTimesExecuted+1;

	gIndexInks := gIndexInks + 1; //Point to the next Bar

END_PROGRAM
```

#### PIDParams.st
```iecst
(* TODO: Add your comment here *)
FUNCTION stPIDParamId
	stPIDParamId:=parPid.rKd + 11 * parPid.rKp + 13 * parPid.rTd + 17 * parPid.rTi;
END_FUNCTION

FUNCTION stPIDParamToMTPIDParameters

//	pidParMeniscus.Gain 			:= parBar.paramsPidMeniscus.rKp;
//	pidParMeniscus.IntegrationTime 	:= parBar.paramsPidMeniscus.rTi;
//	pidParMeniscus.DerivativeTime 	:= parBar.paramsPidMeniscus.rKd;
//	pidParMeniscus.FilterTime 		:= parBar.paramsPidMeniscus.rTd;

	MTPIDparam.Gain 			:= pidParam.rKp;
	MTPIDparam.IntegrationTime 	:= pidParam.rTi;
	MTPIDparam.DerivativeTime 	:= pidParam.rKd;
	MTPIDparam.FilterTime 		:= pidParam.rTd;

	stPIDParamToMTPIDParameters := TRUE;

END_FUNCTION
```

#### powPrintHeads.st
```iecst
ACTION powPrintHeads:

	inks.signals.out.xOutPowPrintHead:=inks.ordersSw.xPowPrintHead AND NOT inks.Al.xAlrPrintHeadPsuFailure AND NOT inks.Al.xAlrPrintHeadsChillerStopped;

END_ACTION
```

#### pressPosAcceleration.st
```iecst
ACTION pressPosAcceleration:

	blink1s(T_Blink:= T#250ms);

	IF NOT EDGEPOS(blink1s.Out) THEN
		RETURN;
	END_IF

	IF rSetPointFillingPump < rOrderBPositiveStart THEN
		(*UP*)
		IF rOrderBPositiveStart - rSetPointFillingPump <= parBar.rAccelerationFillingPump THEN
			rOrderBPositiveStart := rSetPointFillingPump;
		ELSE
			rOrderBPositiveStart := rOrderBPositiveStart - parBar.rAccelerationFillingPump;
		END_IF;
	ELSIF rSetPointFillingPump > rOrderBPositiveStart THEN
		(*DOWN*)
		IF rSetPointFillingPump - rOrderBPositiveStart <= parBar.rAccelerationFillingPump THEN
			rOrderBPositiveStart := rSetPointFillingPump;
		ELSE
			rOrderBPositiveStart := rOrderBPositiveStart + parBar.rAccelerationFillingPump;
		END_IF;
	END_IF;

	IF mode1 THEN //INKS_STOPPED
		rOrderBPositiveStart:=0.0;
	END_IF

END_ACTION
```

#### reservoirMode.st
```iecst
ACTION reservoirMode:

	//Determine if system is stable or not >= 2  and <= 14
	TON_PressureReservoirStable.IN:= mode4 AND //INKS_STARTED
									xReservoirModeActivated AND NOT inks.commands.xCloseReliefValve AND
									rPressureCollectorPos1 >= lc_rLowPresEnterStable AND
									rPressureCollectorPos1 <= lc_rHighPresEnterStable;
	TON_PressureReservoirStable.PT:= T#1S;
	TON_PressureReservoirStable();

	IF TON_PressureReservoirStable.Q THEN
		xPressureReservoirStable := TRUE;
	END_IF

	IF 	NOT mode4 OR //INKS_STARTED
		rPressureCollectorPos1 > lc_rHighPresExitStable OR
		rPressureCollectorPos1 <= lc_rLowPresExitStable OR
		inks.commands.xCloseReliefValve 						THEN
			xPressureReservoirStable := FALSE;
	END_IF

	//Take care about be sure to have the system stabilized with the valve closed
	TON_TimeAfterCloseReliefValve.IN := NOT xPressureReservoirStable;
	TON_TimeAfterCloseReliefValve.PT := T#2S;
	TON_TimeAfterCloseReliefValve();

	inks.signals.out.xReliefValve:= xPressureReservoirStable AND NOT inks.commands.xCloseReliefValve;
	inks.status.xReservoirMode := xReservoirModeActivated;

END_ACTION
```

#### solenoids.st
```iecst
ACTION solenoids:

	xAuxSolenoidDirect:=inks.status.iDirection = INKSDIR_DIRECT OR
						(inks.status.iDirection = INKSDIR_REVERSE AND NOT TON_Stab2.Q) OR
						(inks.status.iDirection = INKSDIR_STOP AND NOT TON_CloseSole.Q);

	xAuxSolenoidReverse:=(inks.status.iDirection = INKSDIR_DIRECT AND NOT TON_Stab1.Q) OR
						inks.status.iDirection = INKSDIR_REVERSE OR
						(inks.status.iDirection = INKSDIR_STOP AND NOT TON_CloseSole.Q);

	IF inks.status.iDirection = INKSDIR_STOP THEN
		AuxiliarSolenoid := FALSE;
	ELSIF inks.status.iDirection = INKSDIR_DIRECT OR inks.status.iDirection = INKSDIR_REVERSE THEN
		AuxiliarSolenoid := TRUE;
	END_IF

	inks.signals.out.xSolenoid1:= xAuxSolenoidDirect AND AuxiliarSolenoid ;
	inks.signals.out.xSolenoid4:= xAuxSolenoidDirect;

	inks.signals.out.xSolenoid2:= xAuxSolenoidReverse;
	inks.signals.out.xSolenoid3:= xAuxSolenoidReverse AND AuxiliarSolenoid ;

	iStabSoleW:=parBar.iStabSole;
	iDisablePidW:=parBar.iDesahPid;
	iCloseSoleW:=parBar.iCloseSole;

	IF iStabSoleW < 200 THEN iStabSoleW := 200; END_IF
	IF iDisablePidW < 250 THEN iDisablePidW := 250; END_IF

	TON_Stab1(	IN:= inks.status.iDirection = INKSDIR_DIRECT,
				PT:= INT_TO_TIME(iStabSoleW));

	TON_Stab2(	IN:= inks.status.iDirection = INKSDIR_REVERSE,
				PT:= INT_TO_TIME(iStabSoleW));

	TON_CloseSole(	IN:= inks.status.iDirection = INKSDIR_STOP,
					PT:= INT_TO_TIME(iCloseSoleW));

	TON_StabSolPid1Neg(IN:= inks.status.iDirection = INKSDIR_REVERSE,
						PT:= INT_TO_TIME(iDisablePidW) );	//This value [3] is to have less time Hold the negative pump

	TON_StabSolPid1Pos(IN:= TON_StabSolPid1Neg.IN,
						PT:= INT_TO_TIME(iDisablePidW));

	TON_StabSolPid2Neg(IN:= mode4 AND //INKS_STARTED
							(iInkPreviousState = INKS_AUTO_REVERSEFLOW OR iInkPreviousState = INKS_MANUAL_REVERSEFLOW),
						PT:= INT_TO_TIME(iDisablePidW) );  //This value [3] is to have less time Hold the negative pump

	TON_StabSolPid2Pos(IN:= TON_StabSolPid2Neg.IN,
						PT:= INT_TO_TIME(iDisablePidW));

END_ACTION
```

#### startUp.st
```iecst
ACTION startUp:

	IF EDGEPOS(inks.parameters.StartUp.xActive) THEN
		inks._Internal.Startup.rSetPointMeniscus := inks.parameters.parBar.StartUp.rMeniscus;
		//inks._Internal.Startup.rSetPointPositive := inks.parameters.parBar.StartUp.rPositive;
		SetStartUpStarting;
	END_IF

	//Exit if not active
	IF NOT inks.parameters.StartUp.xActive THEN
		RETURN;
	END_IF

	// Running each inks system timer
	IF ABS(inks.status.rMeniscus - inks._Internal.Startup.rSetPointMeniscus) <= inks.parameters.parBar.StartUp.rMarginToStable THEN
		xStabMeniscus:= TRUE;
	ELSIF tonNotStabInkStartUp.Q THEN
		xStabMeniscus:= FALSE;
	END_IF

	tonStabInkStartUp.IN := xStabMeniscus;
	tonStabInkStartUp.PT := UINT_TO_TIME(inks.parameters.parBar.StartUp.iSecondsStable * 1000);
	tonStabInkStartUp();

	tonUstabInkStartUp.IN := ABS(inks.status.rMeniscus - inks._Internal.Startup.rSetPointMeniscus) > inks.parameters.parBar.StartUp.rMarginToStable;
	tonUstabInkStartUp.PT := t#5m;
	tonUstabInkStartUp();

	tonNotStabInkStartUp.IN := ABS(inks.status.rMeniscus - inks._Internal.Startup.rSetPointMeniscus) > inks.parameters.parBar.StartUp.rMarginToStable;
	tonNotStabInkStartUp.PT := UINT_TO_TIME(inks.parameters.parBar.StartUp.iSecondsUnstable * 1000);
	tonNotStabInkStartUp();

	// Calculate the step
	rMeniscusStartUpStep := (inks.parSw.NegPump.rSetPointMeniscus - inks.parameters.parBar.StartUp.rMeniscus) / inks.parameters.parBar.StartUp.iSteps;

	// Change setpoints if needed
	IF tonStabInkStartUp.Q THEN

		IF ABS(inks.parSw.NegPump.rSetPointMeniscus - inks._Internal.Startup.rSetPointMeniscus) > 0.1 THEN
			// The system still not in final values
			inks._Internal.Startup.rSetPointMeniscus := inks._Internal.Startup.rSetPointMeniscus + rMeniscusStartUpStep;
			tonStabInkStartUp(IN := FALSE); //Resetting the timer
			xStabMeniscus:= FALSE;
		ELSE
			// The system has arrived
			SetStartUpStarted;
			inks.parameters.StartUp.xActive := FALSE;
		END_IF
	END_IF

	IF tonUstabInkStartUp.Q THEN
		// If detected a long unstability, change the set point to avoid stopping or dripping and raise the signal to go to error
		inks.parSw.NegPump.rSetPointMeniscus := inks.parSw.NegPump.rSetPointMeniscus - rMeniscusStartUpStep;
		SetStartUpCancelled;
		inks.parameters.StartUp.xActive := FALSE;
	END_IF

	// If the system is stopped, mark as cancelled
	IF  NOT inks.status.xInksRunning THEN
		SetStartUpCancelled;
		inks.parameters.StartUp.xActive := FALSE;
	END_IF

END_ACTION

ACTION SetStartUpStarting:
	inks.status.AutoStartUp.xStarting := TRUE;
	inks.status.AutoStartUp.xStarted := FALSE;
	inks.status.AutoStartUp.xCancelled := FALSE;
END_ACTION

ACTION SetStartUpStarted:
	inks.status.AutoStartUp.xStarting := FALSE;
	inks.status.AutoStartUp.xStarted := TRUE;
	inks.status.AutoStartUp.xCancelled := FALSE;
END_ACTION

ACTION SetStartUpCancelled:
	inks.status.AutoStartUp.xStarting := FALSE;
	inks.status.AutoStartUp.xStarted := FALSE;
	inks.status.AutoStartUp.xCancelled := TRUE;
END_ACTION
```

#### tempControl.st
```iecst
ACTION tempControl:

		//heating resistor management
	TON_HeaterStarts.IN := inks.status.iInkState = INKS_STARTING OR inks.status.iInkState = INKS_PRIMING ;
	TON_HeaterStarts.PT := T#20S;
	TON_HeaterStarts();

	// (20secs) gc_tiTiempoRetardoActTemp is the delay when InkSystem is starting
	xStartHeating := TON_HeaterStarts.Q OR inks.status.iInkState = INKS_STARTED OR xStateReverseFlow;
	inks.signals.out.xHeatingActive:=xStartHeating;

	//heating resistor tank management
	xStartTankHeating := TON_HeaterStarts.Q OR inks.status.iInkState = INKS_STARTED OR xStateReverseFlow;

	//Automatic Update ParPID
	parPidTemp:=stPIDParamId(parBar.paramsPidTemp);
	xUpdatePidTemp:= parPidTempCopy <> parPidTemp;
	parPidTempCopy:=parPidTemp;
	IF xUpdatePidTemp THEN
		stPIDParamToMTPIDParameters(ADR(parBar.paramsPidTemp), ADR(pidParTemp));
		stPIDParamToMTPIDParameters(ADR(parBar.paramsPidTankTemp), ADR(pidParTempTank));

		iQuantityUpdatePidTemp:=iQuantityUpdatePidTemp+1;
	END_IF;

	//Changing PID for ink heating when is lower than Set Point Temperature
	IF inks.status.Temp.rTemp < rSPtemp - 1.5 THEN
		inks.status.Temp.rPresetValue:= inks.status.Temp.rTemp - ( (rSPtemp - inks.status.Temp.rTemp) * inks.parameters.Temp.rk1Temp);

	ELSIF inks.status.Temp.rTemp > rSPtemp - 1.5 AND inks.status.Temp.rTemp < rSPtemp THEN
		inks.status.Temp.rPresetValue:= inks.status.Temp.rTemp - ( (rSPtemp - inks.status.Temp.rTemp) * inks.parameters.Temp.rk2Temp);

	ELSIF inks.status.Temp.rTemp > rSPtemp AND inks.status.Temp.rTemp < rSPtemp + 1.5 THEN
		inks.status.Temp.rPresetValue:= inks.status.Temp.rTemp - ( (rSPtemp - inks.status.Temp.rTemp) * inks.parameters.Temp.rk3Temp);

	ELSIF inks.status.Temp.rTemp > rSPtemp + 1.5 THEN
		inks.status.Temp.rPresetValue:= inks.status.Temp.rTemp - ( (rSPtemp - inks.status.Temp.rTemp) * inks.parameters.Temp.rk4Temp);

	END_IF

	// PID PID PID PID PID PID PID PID PID PID PID PID PID PID PID PID PID PID PID PID PID PID PID PID PID PID PID PID PID PID
	fb_PID_Temp(Enable:= xStartHeating AND NOT xPidTempTunning,
				PIDParameters:=pidParTemp,
				HoldOut:= inks.status.iDirection = INKSDIR_REVERSE OR inks.Al.xAlrKlixonTriggered,
				MinOut:=0.0,
				MaxOut:=100.0,
				Update:= xUpdatePidTemp,
				SetValue:=rSPtemp,
				ActValue:=inks.status.Temp.rPresetValue
	);
	inks.status.Temp.rDutyCycleTemp:=fb_PID_Temp.Out;
	inks.status.Temp.xEnabledPid := fb_PID_Temp.Enable;

	//When DuctyCyleTemp is upper than supported by Psu then is applied ReductionTempPower factor in all bars
	inks.status.Temp.rDutyCycleTempPowerRed:= inks.status.Temp.rDutyCycleTemp * inks.parameters.Temp.rReductionTempPower;

	IF xStartHeating THEN
		rDutyCycleTempAux:=   inks.status.Temp.rDutyCycleTempPowerRed;
	ELSE
		rDutyCycleTempAux:= 0;
	END_IF

	IF xPidTempTunning AND xStartHeating THEN
		rDutyCycleTempAux:= rDutyCyclePreTune + fbTempTunning.Out;
	END_IF

	fbTempTunning.Enable := xPidTempTunning;
	fbTempTunning();
	fbTempTunning.ActValue:=inks.status.Temp.rTemp;
	inks.status.Temp.xEnabledTunning := xPidTempTunning;

	// Starting the PWM signal in the right moment to avoid all the bars starting at same time
	xStartTempPwm:= timeToStartPWM(iItemNumber:=iBarNumberInBlock, iTotalItems:= inks.parameters.Temp.iBarsWithSamePsu , iTaskCycle:=iPeriode, iMsInCycle:=iMs);
	xEnablePwmTemp:= xStartHeating  AND ( xStartTempPwm OR xEnablePwmTemp) ;

	// PWM PWM PWM PWM PWM PWM PWM PWM PWM PWM PWM PWM PWM PWM PWM PWM PWM PWM PWM PWM PWM PWM PWM PWM
	fb_PWM_Temp(Enable:= xEnablePwmTemp,
				Mode:=mtBASICS_PULSE_BEGINNING,
				DutyCycle:=rDutyCycleTempAux,
				Period:=lc_rCyclePwm,
	);
	inks.signals.out.xOutBarResistance:=fb_PWM_Temp.Out;
	inks.status.Temp.xEnabledPwm := xEnablePwmTemp;
	inks.status.Temp.rDutyCyclePwm := rDutyCycleTempAux;

	//if I'm not working, the relay exit is off.
	IF	NOT xStartHeating OR fb_PID_Temp.HoldOut THEN
		inks.signals.out.xOutBarResistance:= FALSE;
	END_IF

	/////////////////////////TANK HEATER CONTROL////////////////////////////////////////
	tempTankControl;

END_ACTION

ACTION tempTankControl:

	IF NOT inks.parSw.Temp.xTankHeaterEnabled THEN
		inks.status.Temp.xEnabledTankHeater := FALSE;
		inks.signals.out.xOutResistanceTank:=FALSE;
		RETURN;
	END_IF

	IF NOT inks.status.Tank.xMinLevel OR NOT inks.status.xInksRunning OR NOT inks.parSw.Temp.xTankHeaterEnabled OR inks.Al.xAlrHeaterTankPsu OR inks.Al.xAlrHeaterTankReachsMaxTemp THEN
		inks.status.Temp.xEnabledTankHeater := FALSE;
	ELSIF xStartTankHeating THEN
		inks.status.Temp.xEnabledTankHeater := TRUE;
	END_IF

	// PID PID PID PID PID PID PID PID PID PID PID PID PID PID PID PID PID PID PID PID PID PID PID PID PID PID PID PID PID PID
	fb_PID_Tank_Temp(Enable:= inks.status.Temp.xEnabledTankHeater,
					PIDParameters:=pidParTempTank,
					MinOut:=0.0,
					MaxOut:=100.0,
					SetValue:=rSPTempTank,
					ActValue:=inks.status.Temp.rTempTank);
	inks.status.Temp.rDutyCycleTempTank:=fb_PID_Tank_Temp.Out;

	// PWM PWM PWM PWM PWM PWM PWM PWM PWM PWM PWM PWM PWM PWM PWM PWM PWM PWM PWM PWM PWM PWM PWM PWM
	fb_PWM_Temp_Tank(Enable:= fb_PID_Tank_Temp.Enable,
					DutyCycle:=inks.status.Temp.rDutyCycleTempTank, Period:=2.0);

	inks.status.xInkAndPreheatingRunning:= fb_PID_Tank_Temp.Enable;
	inks.signals.out.xOutResistanceTank:=fb_PWM_Temp_Tank.Out;

END_ACTION
```

### Inks Notes.txt - Inks Notes
```
Converted previously genVar by Command
g_xIgnoraAlarmasPorLimpieza >> data.commands.xIgnoreAlarmsInCleaning
```

### Inks.typ - Inks Data definition
```iecst
TYPE
	inksDirections :
		(
		INKSDIR_DIRECT := 1,
		INKSDIR_REVERSE := 2,
		INKSDIR_STOP := 3
		);
	inksStateModes :
		(
		INKS_STOPPED := 1,
		INKS_STARTING := 3,
		INKS_STARTED := 4,
		INKS_MANUAL_REVERSEFLOW := 5,
		INKS_AUTO_REVERSEFLOW := 6,
		INKS_STOPPING := 9,
		INKS_RUNNING_MANUAL := 10,
		INKS_PRIMING := 13,
		INKS_UNDEFINED := 255
		);
	stInksCommands : 	STRUCT
		xOrderCleaning : BOOL; (*Command coming from the Block*)
		xOrderDrip : BOOL; (*This signal must be maintained during the dripping. If the order is falled down, the dripping is finished. Command coming from the Block*)
		xCloseReliefValve : BOOL; (*Command coming from the Block*)
		xErrorRst : BOOL;
		xMute : BOOL;
	END_STRUCT;
	stInksStartUpParams : 	STRUCT
		iSteps : USINT;
		iSecondsStable : UINT; (*Seconds in the window and ready for next step*)
		iSecondsUnstable : UINT; (*Seconds to consider we are out of window*)
		rMeniscus : REAL; (*Valuen in mbar*)
		rMarginToStable : REAL; (*Valuen in mbar. Margin to consider Stable*)
	END_STRUCT;
	stInksDefaultBarParams : 	STRUCT
		rMeniscus : REAL;
		rPositive : REAL;
		rTemp : REAL;
	END_STRUCT;
	stInksOrdersSw : 	STRUCT
		xStartInks : BOOL;
		xPowPrintHead : BOOL;
		xStartManual : BOOL;
		xOrderReverseMan : BOOL;
	END_STRUCT;
	stInksBarParams : 	STRUCT
		paramsPidMeniscus : stPIDParam;
		paramsPidPositive : stPIDParam;
		paramsPidTemp : stPIDParam;
		paramsPidTankTemp : stPIDParam;
		paramsPidMeniscusReservoir : stPIDParam;
		paramsPidPositiveReservoir : stPIDParam;
		rHighPumpLimitNeg : REAL;
		rHighPumpLimitPos : REAL;
		rLowPumpLimitNeg : REAL;
		rLowPumpLimitPos : REAL;
		rAccelerationFillingPump : REAL;
		rSPfillingPumpStarting : REAL;
		iStabSole : INT;
		iDesahPid : INT;
		iCloseSole : INT;
		xTypeTankSensorAnalog : BOOL;
		xTypeTankSensorDigital : BOOL;
		iPowerTempWatt : UINT; (*Power of the main heater in the bar*)
		rVacuumSensorSpan : REAL; (*Span of the sensor in mBar*)
		rVacuumSensorOffset : REAL; (*Value in mBar of the minimum value of the sensor*)
		iTimeToActiveDcErrorAlarm : TIME;
		Default : stInksDefaultBarParams;
		StartUp : stInksStartUpParams;
		zFree : ARRAY[0..3]OF USINT;
	END_STRUCT;
	stInksConstantsToSw : 	STRUCT
		tiDripTimeMin : TIME;
		tiDripTimeMax : TIME;
	END_STRUCT;
	stInksParametersSwNegPump : 	STRUCT
		rSetPointMeniscus : REAL; (*Meniscus SetPoint in mbar*)
		rSetPointManual : REAL;
		rLimitMeniscusDiffWarning : REAL;
		rUpperLimMeniscusCritical : REAL;
		rLowerLimMeniscusCritical : REAL;
	END_STRUCT;
	stInksParametersSwPosPump : 	STRUCT
		rSetPoint : REAL; (*Value in mbar*)
		rSetPointManual : REAL;
	END_STRUCT;
	stInksParametersSwTemp : 	STRUCT
		rSetPointTemp : REAL; (*Value in ºC*)
		rSetPointTempMaintenance : REAL; (*Value in ºC. Temp SP to be used when maintenance mode activated*)
		xTankHeaterEnabled : BOOL := FALSE;
	END_STRUCT;
	stInksParametersSwConfig : 	STRUCT
		iMappingBar : UINT;
		iInkType : INT := 1; (*Default value is 1, *)
		iPrintHeadType : INT; (*Printhead type xBar (0=ERROR, 1=TTEC, 2=Seiko, 3=XAAR, 4=Dimatix, 5=TTEC_XL, 6=X_GS40, 7=XAAR2001, 8=XAAR2001GS40, 9=SEIKOW, 10=SeikoL)*)
	END_STRUCT;
	stInksParametersSw : 	STRUCT
		xActMaintenanceMode : BOOL; (*Active when bar is in maintenance mode. To read parSw "rSetPointTempMaintenance" instead of "rSetPointTemp"*)
		xActTestMode : BOOL;
		xEnabledBarToPrint : BOOL;
		xOnReverseCapped : BOOL;
		xOnReverseCleaning : BOOL;
		xReverseOnManual : BOOL := FALSE; (*Activate reverser Flow in Manual activation of the Inks*)
		xColorLoadedInJob : BOOL; (*Active when bar is enabled to print and is used by current loaded job*)
		tiReverseManual : TIME;
		tiDripTime : TIME; (*Time dripping the Bar*)
		iInkEnabledPrintHeads : INT; (*Quantity of printheads enabled*)
		iInkConsumption : INT; (*Picoliters/m2*)
		Config : stInksParametersSwConfig;
		NegPump : stInksParametersSwNegPump;
		PosPump : stInksParametersSwPosPump;
		Temp : stInksParametersSwTemp;
	END_STRUCT;
	stInksParametersNegPump : 	STRUCT
		rSetPointPrimingStarting : REAL := 30; (*DC thres in Positive pump to change SP applied to PID in PrimingSystems*)
		rDCPriming : REAL := 10;
	END_STRUCT;
	stInksParametersPosPump : 	STRUCT
		rSetPointPrimingStarting : REAL := 10; (*DC thres in Positive pump to change SP applied to PID in PrimingSystems*)
		rDCThresholdPriming : REAL := 30.0; (*DC thres in Positive pump to change SP applied to PID in PrimingSystems*)
		rDCPriming : REAL := 50;
	END_STRUCT;
	stInksParametersTemp : 	STRUCT
		rReductionTempPower : REAL := 1.0; (*Not reducing power by default.*)
		rk1Temp : REAL := 0; (*Coefficient k1 applied to PID*)
		rk2Temp : REAL := 6; (*Coefficient k2 applied to PID*)
		rk3Temp : REAL := 2; (*Coefficient k3 applied to PID*)
		rk4Temp : REAL := 4; (*Coefficient k4 applied to PID*)
		iBarsWithSameBlock : UINT;
		iBarsWithSamePsu : UINT;
	END_STRUCT;
	stInksParametersPriming : 	STRUCT
		xSystemNeedsPriming : BOOL;
		rThresholdPressure : REAL := 2; (*DC thres in Positive pump to change SP applied to PID in PrimingSystems*)
	END_STRUCT;
	stInksParametersChiller : 	STRUCT
		Status : ChillerStatus_enum; (*Chiller status*)
		iIndex : USINT;
	END_STRUCT;
	stInksParametersStartUp : 	STRUCT
		xActive : BOOL; (*StartUp is active. This is activated remotely, and reseted remotely if cancelled, or reseted internally if finished*)
	END_STRUCT;
	stInksParameters : 	STRUCT
		parBar : {REDUND_UNREPLICABLE} stInksBarParams;
		StartUp : stInksParametersStartUp;
		tiDripTimeMax : TIME; (*Max dripping time of the started bars in the same block*)
		iTimeStopping : INT;
		xDebugMode : BOOL := FALSE;
		xReservoirMode : BOOL;
		iTimeChangeSPInRev : UINT := 6; (*Delay to change SP applied to PID of negative pump*)
		NegPump : stInksParametersNegPump;
		PosPump : stInksParametersPosPump;
		Temp : stInksParametersTemp;
		Priming : stInksParametersPriming;
		xEnabledTachoSignals : BOOL; (*Define if the system has Tacho signal in the pumps*)
		xBlockInCap : BOOL := FALSE; (*Ink has to know when block is capped to apply reverse Idle (60 sec of revese every 30 min) when Idle checkbos is enabled from GUI*)
		xBlockInPrint : BOOL := FALSE; (*Ink has to know when block is print to check the excesive diferential temperature to print. Only in print and automatic state.*)
		InksChiller : stInksParametersChiller;
		PrintheadsChiller : stInksParametersChiller;
	END_STRUCT;
	stInksStatusTemp : 	STRUCT
		xEnabledPid : BOOL; (*Enable the Pid FB*)
		xEnabledPwm : BOOL; (*Enable the Pwm FB*)
		xEnabledTunning : BOOL; (*Enable the Tunning FB*)
		rDutyCyclePwm : REAL; (*Duty Cycle for Temperature control directly to the PWM FB*)
		rDutyCycleTempPowerRed : REAL; (*Duty Cycle for Temperature control with the Power Reduction due to less power in PSU than in heaters*)
		xEnabledTankHeater : BOOL; (*It informs about tank heater status*)
		rDutyCycleTempPowerRedTank : REAL; (*Dutty Cycle Heater Tank. Added this status. It informs to datalogger.*)
		rDutyCycleTempTank : REAL; (*Dutty Cycle Heater Tank*)
		rDutyCycleTemp : REAL;
		rPresetValue : REAL; (*Temperature value when PID is agressive*)
		rTemp : REAL;
		rTempTank : REAL;
	END_STRUCT;
	stInksStatusNegPump : 	STRUCT
		rDutyCycleNegative : REAL;
		rSpeedNeg : REAL; (*Speed in rpm*)
		rCurrent : REAL; (*Current consumption measured by PLC*)
	END_STRUCT;
	stInksStatusPosPump : 	STRUCT
		rDutyCycleFilling : REAL;
		rSpeedPos : REAL; (*Speed in rpm*)
		rSetPointPos : REAL;
		rCurrent : REAL; (*Current consumption measured by PLC*)
	END_STRUCT;
	stInksStatusReverse : 	STRUCT
		xOnReverseAuto : BOOL;
		xOnReverseCleaning : BOOL := FALSE;
		xOnReverseCapped : BOOL := FALSE;
		xReverseOnManual : BOOL;
		xReverseMan : BOOL := FALSE;
		xReverseManFinished : BOOL := FALSE;
		xStartOnReverseCapped : BOOL := FALSE;
		xStartOnReverseCappedCycle : BOOL := FALSE;
	END_STRUCT;
	stInksStatusTank : 	STRUCT
		iStatusTankDigital : INT;
		iDipositLevel : INT;
		xMaxLevel : BOOL; (*There is more ink than the MAXIMUM sensor level. The MAXIMUM sensor level is active*)
		xCloseToMinLevel : BOOL; (*There is more ink than the MINIMUM sensor level. The MINIMUM sensor level is active but unstable*)
		xMinLevel : BOOL; (*There is more ink than the MINIMUM sensor level. The MINIMUM sensor level is active*)
	END_STRUCT;
	stInksStatusAutoStartUp : 	STRUCT
		xStarting : BOOL;
		xCancelled : BOOL;
		xStarted : BOOL;
	END_STRUCT;
	stInksStatus : 	STRUCT
		Temp : stInksStatusTemp;
		NegPump : stInksStatusNegPump;
		PosPump : stInksStatusPosPump;
		Tank : stInksStatusTank;
		iDirection : inksDirections;
		AutoStartUp : stInksStatusAutoStartUp;
		tiDriptime : TIME;
		xDripping : BOOL;
		iInkStateSw : INT;
		iInkState : inksStateModes;
		tiInReverseManual : TIME; (*Time in reverse Manual*)
		rVacuum1 : REAL; (*Vacuum at Positive in mbar*)
		rVacuum2 : REAL; (*Vacuum at Negative  in mbar*)
		rMeniscus : REAL;
		rDeltaPressure : REAL;
		xInkAndPreheatingRunning : BOOL;
		xInksRunning : BOOL;
		xReservoirMode : BOOL := FALSE;
		Reverse : stInksStatusReverse;
		xUnstableInkState : BOOL;
		startChangeSPInDelta : BOOL;
		xColorLoadedInJob : BOOL;
		xEnabledBarToPrint : BOOL;
		xActTestMode : BOOL;
		xActMaintenanceMode : BOOL;
		xBarInstalled : BOOL;
	END_STRUCT;
	stInksAlarmsList : 	STRUCT
		xAlrBrokenMeniscus : BOOL;
		xAlrDiffInCtrlTemp : BOOL;
		xAlrDiffVacuum : BOOL;
		xAlrInksRunnig : BOOL;
		xAlrLevelSensorError : BOOL;
		xAlrNoInkNoCleanManif : BOOL;
		xAlrNoRecircStop : BOOL;
		xAlrNoRecirculation : BOOL;
		xAlrOverPressure : BOOL;
		xAlrPumpsDCError : BOOL;
		xAlrStopRecircNoInk : BOOL;
		xAlrTankDigitalSensorsError : BOOL;
		xAlrTankEmpty : BOOL;
		xAlrTankCloseToEmpty : BOOL;
		xAlrTankToFillIn : BOOL;
		xAlrIncoherTempHeat : BOOL;
		xAlrTempSensor : BOOL;
		xAlrTempTankSensor : BOOL;
		xAlrDifCtrlTempExcessive : BOOL;
		xAlrDiffInCtrlTempTank : BOOL;
		xAlrIncoherTempTank : BOOL;
		xAlrVacuum1 : BOOL;
		xAlrVacuum2 : BOOL;
		xAlrVacuumSensor1 : BOOL;
		xAlrVacuumSensor2 : BOOL;
		xAlrKlixonTriggered : BOOL;
		xAlrPrintHeadPsuFailure : BOOL := FALSE;
		xAlrHeaterTankPsu : BOOL;
		xAlrHeaterTankReachsMaxTemp : BOOL;
		xAlrHeaterReachsMaxTemp : BOOL;
		xAlrHeaterOutFault : BOOL; (*Alarm to report PLC output to bar heater*)
		xAlrMaintenanceModeActive : BOOL;
		xHeaterOff : BOOL; (*Chiller is on and heater DC of the bar is 0% for > 120s NOZOMITWO-1410*)
		xAlrPrintHeadsChillerStopped : BOOL; (*The chiller for Printheads is stopped and the printheads with power. Power to Printheads is removed automatically*)
	END_STRUCT;
	stInksSignalsOut : 	STRUCT
		xSolenoid1 : BOOL;
		xSolenoid2 : BOOL;
		xSolenoid3 : BOOL;
		xSolenoid4 : BOOL;
		iDutyCycleNegative : INT;
		iDutyCycleFilling : INT;
		xOutPowPrintHead : BOOL;
		xOutBarResistance : BOOL;
		xOutResistanceTank : BOOL;
		xHeatingActive : BOOL;
		xReliefValve : BOOL;
	END_STRUCT;
	stInksSignalsIn : 	STRUCT
		iInTankLevel : INT;
		xMinLevel : BOOL;
		xMaxLevel : BOOL;
		xOverpressure : BOOL;
		xTempSensorError : BOOL;
		xVacuum1SensorError : BOOL;
		xVacuum2SensorError : BOOL;
		xTempTankSensorError : BOOL;
		xInkLevelTankSensorError : BOOL;
		iTemperatureRaw : INT;
		iTemperatureTankRaw : INT;
		iVacuum1Raw : INT;
		iVacuum2Raw : INT;
		iTachNegative : UINT;
		iTachFilling : UINT;
		xKlixonTriggered : BOOL;
		xConnected : BOOL; (*Feedback signal of electrical connection. Bar terminal strp connected*)
		xPrintHeadsPsuOK : BOOL := FALSE;
	END_STRUCT;
	stInksInternal : 	STRUCT
		Startup : stInksInternalStartup;
	END_STRUCT;
	stInksInternalStartup : 	STRUCT
		rSetPointMeniscus : REAL; (*Meniscus SetPoint in mbar*)
	END_STRUCT;
	stInksSignals : 	STRUCT
		in : stInksSignalsIn;
		out : stInksSignalsOut;
	END_STRUCT;
	stInks : 	STRUCT
		commands : stInksCommands;
		ordersSw : stInksOrdersSw;
		parameters : stInksParameters;
		parSw : stInksParametersSw;
		status : stInksStatus;
		signals : stInksSignals;
		Al : stInksAlarmsList;
		AlSummary : stEFI_AlarmSummary;
		_Internal : stInksInternal;
	END_STRUCT;
END_TYPE
```

### Inks Docu.txt - How to use it
```
#################################################################################
#################################################################################
#																				#
#			GENERAL USE OF Inks										     		#
#																				#
# 	To use this INKs unit, some general variables are needed:					#
#################################################################################

#################################################################################
#################################################################################
#																				#
#			¡¡¡IMPORTANT!!!!													#
# 	Review InksCtrl and 														#
# 																				#
#																				#
#################################################################################
```

### InksCtrl.md - Inks package actuators behaviour
```markdown
| Doc Version | Description                       | Date       | Resp       |
| ----------- | --------------------------------- | ---------- | ---------- |
| 1.0         | Create doc baed in actual package | 08/05/2024 | J. Alarcón |
|             |                                   |            |            |
|             |                                   |            |            |

# Actuators behaviour

Check Diagram states document

| **Actuator**   | **STOPPED**                        | **STARTING**                                                     | **STARTED**                       | **MANUAL_REVERSFLOW**             | **AUTO_REVERSEFLOW**              | **STOPPING**                       | **RUNNING_MANUAL**                | **PRIMING**                       |
| -------------- | ---------------------------------- | ---------------------------------------------------------------- | --------------------------------- | --------------------------------- | --------------------------------- | ---------------------------------- | --------------------------------- | --------------------------------- |
| xSolenoid1     | OFF                                | ON                                                               | ON                                | OFF (with Delay parBar.iStabSole) | OFF (with Delay parBar.iStabSole) | OFF                                | ON                                | ON                                |
| xSolenoid 2    | OFF (with Delay parBar.iCloseSole) | OFF (with Delay)                                                 | OFF (with<br> Delay)              | ON (with Delay parBar.iStabSole)  | ON (with Delay parBar.iStabSole)  | OFF (with Delay parBar.iCloseSole) | OFF (with<br> Delay)              | OFF (with<br> Delay)              |
| xSolenoid 3    | OFF                                | OFF (with Delay parBar.iStabSole)                                | OFF (with Delay parBar.iStabSole) | ON                                | ON                                | OFF                                | OFF (with Delay parBar.iStabSole) | OFF (with Delay parBar.iStabSole) |
| xSolenoid 4    | OFF (with Delay parBar.iCloseSole) | ON                                                               | ON                                | OFF (with Delay parBar.iStabSole) | OFF (with Delay parBar.iStabSole) | OFF (with Delay parBar.iStabSole)  | ON                                | ON                                |
| xReliefValve   | CLOSE                              | xPressureReservoirStable AND NOT inks.commands.xCloseReliefValve | CLOSE                             | CLOSE                             | CLOSE                             | CLOSE                              | CLOSE                             | CLOSE                             |
| PosPump        | 0.0                                | PID                                                              | PID                               | PID                               | PID                               | 0.0                                | parSw.PosPump.rSetPointManual     | rDCPriming                        |
| NegPump        | 0.0                                | PID                                                              | PID                               | PID                               | PID                               | 0.0                                | parSw.NegPump.rSetPointManual     | rDCPriming                        |
| BarResistance  | OFF                                | PID+PWM                                                          | PID+PWM                           | OFF                               | OFF                               | OFF                                | OFF                               | PID+PWM                           |
| TankResistance | OFF                                | PID+PWM                                                          | PID+PWM                           | PID+PWM                           | PID+PWM                           | OFF                                | OFF                               | PID+PWM                           |

## PID set point values

|                                 | STARTING                                                                             | STARTED                                                                              | MANUAL_REVERSFLOW                                                                                                          | AUTO_REVERSEFLOW                                                                                                           |
| ------------------------------- | ------------------------------------------------------------------------------------ | ------------------------------------------------------------------------------------ | -------------------------------------------------------------------------------------------------------------------------- | -------------------------------------------------------------------------------------------------------------------------- |
| Meniscus  pressure SP (NegPump) | IF automatic start +up THEN Internal value (25) ELSE parSw.NegPump.rSetPointMeniscus | IF automatic start +up THEN Internal value (25) ELSE parSw.NegPump.rSetPointMeniscus | 25 if DeltaPressure <= 20 other case: IF automatic start +up THEN Internal value (25) ELSE parSw.NegPump.rSetPointMeniscus | 25 if DeltaPressure <= 20 other case: IF automatic start +up THEN Internal value (25) ELSE parSw.NegPump.rSetPointMeniscus |
| Filling  pressure SP (PosPump)  | inks.parSw.PosPump.rSetPoint                                                         | inks.parSw.PosPump.rSetPoint                                                         | -15 if DeltaPressure <= 20 Other case: inks.parSw.PosPump.rSetPoint                                                        | -15 if DeltaPressure <= 20 Other case: inks.parSw.PosPump.rSetPoint                                                        |
```

### Program Logical/ExtPack/InksCtrl/InksSim/InksSim_v1/InksSim (IEC) - Simulation of an InkSystem

#### Main.st - Init, cyclic, exit code
```iecst
PROGRAM _INIT
	(* Insert code here *)
	simTemp.rA:= 0.2;
	simTemp.rB:= 0.01;
	simTemp.rInitialValue:= 200;
	simTemp.rMinValue:= 150;
	simTemp.rMaxValue:= 600;

	simPresPos.rA:= 1.8;
	simPresPos.rB:= 0.008;
	simPresPos.rInitialValue:= 16383;
	simPresPos.rMinValue:= 13000;
	simPresPos.rMaxValue:= 25000;

	simPresNeg.rA:= -20;
	simPresNeg.rB:= -0.1;
	simPresNeg.rInitialValue:= 16383;
	simPresNeg.rMinValue:= 8000;
	simPresNeg.rMaxValue:= 25000;

	FOR iInksSimIndex:= 1 TO MAX_LAST_INK DO
		SimInks ACCESS ADR(gSimInks[iInksSimIndex]);
		SimInks.Parameters.TankValuePercent := 50.0;
	END_FOR

END_PROGRAM

PROGRAM _CYCLIC

	Inks ACCESS ADR(gInks[iInksSimIndex]);
	SimInks ACCESS ADR(gSimInks[iInksSimIndex]);

	//Define here the parameters modified at the first execution
	IF NOT xStarted THEN
		//Inks.parSw.Temp.rSetPointTemp:=30.0;
		xStarted:=TRUE;
	END_IF

	IF EDGEPOS(Inks.status.iInkState = INKS_STARTING) THEN
		IF gMachine.St.Mode.xStartUp THEN
			simPresPos.rNewPresentValue:=14500;
			simPresNeg.rNewPresentValue:=13000;
		ELSE
			simPresPos.rNewPresentValue:=16500;
			simPresNeg.rNewPresentValue:=13000;
		END_IF
		simPresPos.xUseNewValue:=TRUE;
		simPresNeg.xUseNewValue:=TRUE;
	END_IF

	tonNotHeating.IN := NOT Inks.signals.out.xOutBarResistance;
	tonNotHeating.PT := T#2500ms;
	tonNotHeating();
	//If not really heating, not increase temperature in simulation
	IF tonNotHeating.Q THEN
		simTemp.rActionControl:=0;
	ELSE
		simTemp.rActionControl:=Inks.status.Temp.rDutyCycleTemp;
	END_IF
	simTemp();
	Inks.signals.in.iTemperatureRaw := REAL_TO_INT(simTemp.rPresentValue);

	simPresPos.rActionControl:= Inks.status.PosPump.rDutyCycleFilling * 10;
	simPresPos();
	Inks.signals.in.iVacuum1Raw := REAL_TO_INT(simPresPos.rPresentValue);

	simPresNeg.rActionControl:= Inks.status.NegPump.rDutyCycleNegative * 10;
	simPresNeg();
	Inks.signals.in.iVacuum2Raw := REAL_TO_INT(simPresNeg.rPresentValue);

	// Code in Inks
	// fbFilterLevelSensor.In:=(((INT_TO_REAL(inks.signals.in.iInTankLevel-16383)*1500)/16384.0)),	WindowLength:=60);
	// rTankLevelmm:= fbFilterLevelSensor.Out;
	// rTankLevelPercent:= LIMIT(0, (rTankLevelmm/2.35), 100);
	Inks.signals.in.iInTankLevel := REAL_TO_INT((SimInks.Parameters.TankValuePercent * 2.35 * 16384 / 1500) + 16383);

	//Go to the next element
	iInksSimIndex := iInksSimIndex +1;

END_PROGRAM

PROGRAM _EXIT
	(* Insert code here *)

END_PROGRAM
```

### Program Logical/ExtPack/InksCtrl/InksSim/InksSim_v1/InitInksSim (IEC)

#### InitInks.st
```iecst
PROGRAM _CYCLIC
	iInksSimIndex := 1;
END_PROGRAM
```

### InkSim.typ
```iecst
TYPE
	SimInkCommands_typ : 	STRUCT
		xCommand : BOOL; (*New command to implement*)
	END_STRUCT;
	SimInkParameters_typ : 	STRUCT
		TankValuePercent : REAL; (*Tank Value percent desired*)
	END_STRUCT;
	SimInk_typ : 	STRUCT
		Commands : SimInkCommands_typ;
		Parameters : SimInkParameters_typ;
	END_STRUCT;
END_TYPE
```

### Block.typ
```iecst
TYPE
	Block_States_enum :
		(
		BLOCK_STOPPED,
		BLOCK_STOPPING,
		BLOCK_MANUAL,
		BLOCK_AUTO
		);
	Block_Position_enum :
		(
		BLOCKP_UNDEFINED,
		BLOCKP_IN_CAP,
		BLOCKP_IN_PRINT,
		BLOCKP_IN_CLEAN,
		BLOCKP_CLEANING,
		BLOCKP_GOING_TO_CAP,
		BLOCKP_GOING_TO_PRINT,
		BLOCKP_GOING_TO_CLEAN,
		BLOCKP_HOMING_ICLA,
		BLOCKP_HOMING_BAR
		);
	StBlock_Outputs : 	STRUCT
		xTrayOut : BOOL;
		xTrayIn : BOOL;
		xVenturi : BOOL;
		xShotLine1 : BOOL; (*Output For InstantPrint/ContinuousPrint signal from PLC to Carriage*)
		xShotLine2 : BOOL; (*Output For InstantPrint/ContinuousPrint signal from PLC to Carriage*)
		xEnableDobleShot : BOOL; (*Review*)
		xEnableDrive : BOOL;
		xEnableIclaSI : BOOL;
		xEnableCurtain : BOOL;
		xCleaningWaterPump : BOOL; (*Water Pump to Celaning PrintHeads*)
		xWastedInkTankPump : BOOL; (*Pump to remove wasted ink from wasted ink's tank*)
		xCappingWaterPump : BOOL; (*Water Pump to Celaning PrintHeads*)
		xDegasser : BOOL;
		xTurbine : BOOL; (*Cleanning by turbine order*)
	END_STRUCT;
	StBlock_Log : 	STRUCT
		diMoveARelCounter : DINT;
		diMoveAbsCounter : DINT;
		diHomingsNumber : DINT;
	END_STRUCT;
	StBlock_Alarms : 	STRUCT
		xAlrSafetySystemInBlock : BOOL; (*CriticalAlarm*)
		xAlrDif : BOOL; (*CriticalAlarm*)
		xAlrTempPowerSupply : BOOL; (*Warning:Heater Power Supply Failure*)
		xAlrPHPowerSupply : BOOL; (*Warning:Print Head Power Supply Failure*)
		xAlrDriveProtection : BOOL; (*CriticalAlarm*)
		xAlAirVenturi : BOOL; (*StopAlarm*)
		xModuleTemp01 : BOOL; (*CriticalAlarm*)
		xModuleTemp02 : BOOL; (*CriticalAlarm*)
		xModuleTemp03 : BOOL; (*CriticalAlarm*)
		xModuleTemp04 : BOOL; (*Critical Alarm*)
		xSiUnitPowerOff : BOOL; (*CriticalAlarm*)
		xAlrComSiUnit : BOOL; (*CriticalAlarm*)
		xAlCleanInterrupt : BOOL; (*StopAlarm*)
		xAlrCleanMotor : BOOL; (*CriticalAlarm *)
		xAlrCleanMtrNoRef : BOOL; (*CriticalAlarm *)
		xAlrComCleanMtr : BOOL; (*CriticalAlarm *)
		xAlrDecreaseCleanOffset : BOOL; (*Warning*)
		xAlrIncoherPositCleanMtr : BOOL; (*CriticalAlarm *)
		xAlrEnabCleanMtrDiffLvL : BOOL; (*CriticalAlarm *)
		xAlrTraySensor : BOOL; (*CriticalAlarm *)
		xAnyDriveAlarmLimitMax : BOOL; (*CriticalAlarm *)
		xAlrBarMtrNoRef : BOOL; (*CriticalAlarm *)
		xAlrCleanSensor : BOOL; (*CriticalAlarm                 L59,LC Barras*)
		xAlrComBarMtr : BOOL; (*CriticalAlarm *)
		xExitCleaningCycle : BOOL; (*Silvia*)
		xAnyVerticalDriveAlarm : BOOL; (*CriticalAlarm *)
		xAnyIclaAlarm : BOOL; (*CriticalAlarm *)
		xAlrNoTrayInServoNoHomed : BOOL; (*Warning. Derived alarm*)
		xAlrRearSafety : BOOL; (*Rear Door Open Alarm*)
		xAlrFrontSafety : BOOL; (*Front Door Open Alarm*)
		xAlrFrontEmergencyStop : BOOL;
		xAlrRearEmergencyStop : BOOL;
		xAlrFrontCurtain : BOOL;
		xAlrCrossSensorDetectBottom : BOOL;
		xAlBarMotorPowerOff : BOOL;
		xAlrReferenceIncoherence : BOOL; (*CriticalAlarm*)
		xAlrRearSafetyCircuit : BOOL;
		xAlrFrontSafetyCircuit : BOOL;
		xAlrBlockReachedMaxPosition : BOOL;
		xNoActionDangerCollision : BOOL; (*Some sensor signal not  OK, so no movement allowed*)
		xAlrWaterPumpPresure : BOOL; (*Pump working but not pressure measured. Alarm non Autoreset*)
		xAlrEmptyWaterTank : BOOL;
		xAlrWtrPresSensBroken : BOOL;
		xAlrBarsOut : BOOL;
		xBarMotorTemp : BOOL; (*Warning: Bar Motor Temperature Too Hot*)
		xBarDriverTemp : BOOL; (*Warning: Bar Driver Temperature Too Hot*)
		xAlrCheckHomingSensor : BOOL; (*Warning: Bar Homing Sensor Maybe Broken*)
		xAlrLogicEmergencyStop : BOOL; (*Emergency button pushed without diferenciating front or rear. Calculated from NOT SafetyOK and everything ready (doors and lightCourtains)*)
		xAlrEmergencyStop : BOOL; (*Any Emergency button pushed. Aggregated alarm*)
		xAlrCappingWaterTankEmpty : BOOL;
		xAlrCappingWaterNotRecirc : BOOL; (*Emergency button pushed without diferenciating front or rear*)
		xAlrControllerNotReady : BOOL; (*Critical: Controller of the Drive not Ready. Usually motor not conected to drive*)
		xAlrOverTorque : BOOL;
		xWrnOverTorq : BOOL; (*Warning: Belt Over Torque*)
		xCleanMotorControllerNotReady : BOOL; (*Waiting for enable input (STO_A, STO_B)*)
	END_STRUCT;
	stBlock_commandsManual : 	STRUCT
		xManBarsUp : BOOL; (*Command just in manual mode*)
		xManBarsDown : BOOL; (*Command just in manual mode*)
		xManIclaForward : BOOL; (*Command just in manual mode*)
		xManIclaBack : BOOL; (*Command just in manual mode*)
		xManTrayOut : BOOL; (*Command just in manual mode*)
		xManTrayIn : BOOL; (*Command just in manual mode*)
		xManVenturi : BOOL; (*Command just in manual mode*)
		xManWaterSpurt : BOOL; (*Command just in manual mode*)
		xManCappingWaterPump : BOOL; (*Command just in manual mode*)
		xManWastePump : BOOL; (*Command just in manual mode*)
		xToPrintPosition : BOOL; (*EDGE Command just in Man mode. Sends the block to PrintPosition if previously in Cap*)
	END_STRUCT;
	stBlock_commands : 	STRUCT
		Mode : StGeneral_States_Mode;
		StateMode : enumEFI_GenMachineState; (*commands to block*)
		AutoMode : stEFI_MachineAutoModes; (*commands to inform belt*)
		Manual : stBlock_commandsManual;
		xDripControl : BOOL; (*internal orders in structure? Tthat sould be internal variables as orders. TOJMH: when? *)
		xBarHomeOrder : BOOL; (*State Command just in manual mode*)
		xIclaHomeOrder : BOOL; (*Command just in manual mode*)
		xIclaHomeOrderInterrupt : BOOL; (*Command just in manual mode*)
		xToPrint : BOOL; (*Command just in AUTO mode*)
		xToCap : BOOL; (*Command just in AUTO mode*)
		xToCleanPosition : BOOL; (*EDGE Command just in Man mode. Sends the block to CleanPosition if previously in Cap*)
		xToPrintLab : BOOL; (*EDGE Command. Reseted manually in Block*)
		xToCapLab : BOOL; (*EDGE Command. Reseted manually in Block*)
		xStartToCleanOrder : BOOL; (*EDGE. Reseted by Block. Command just in AUTO mode: The machine raises*)
		xInksOrderCleaning : BOOL; (*Command just in AUTO mode: to activate reverse flow in cap position (automatic before drip and every 30 min)*)
		xMute : BOOL; (*Command Bool mute sound*)
		xReset : BOOL; (*Command Bool Reset*)
		xEnableCleaningWithWater : BOOL; (*Command Bool Enable Cleaning Water Proces*)
		xCleanStop : BOOL; (*Comand to Stop Clean*)
		xForcePreprintingPos : BOOL; (*Comand to Force preprinting position*)
		xForceCleanDelay : BOOL; (*Comand to Clean Block With Delay*)
		xForceCleanNoDelay : BOOL; (*Comand to Clean Block Without Delay*)
	END_STRUCT;
	StBlock_Parameters_Inks : 	STRUCT
		iMaxPSUwattsForBars : UINT := 200; (*This parameter allows changes on PSU max to calculate different factor redutor. Value in watts*)
		iMaxBlockPrintBars : USINT := 6; (*To allow indentify if the bars belongs to the block*)
		iMaxMachinePrintBars : USINT := 12; (*Interger is compared with integers, it avoids warning. This var is used but is pending to implement limits.... take care!!*)
		xTankHeatEnabled1 : BOOL := FALSE; (*Bar 1, 2, 3 or 4 have tank heater enabled*)
		xTankHeatEnabled2 : BOOL := FALSE; (*Bar 5, 6, 7, or 8 have tank heater enabled*)
	END_STRUCT;
	StBlock_Parameters_Icla : 	STRUCT
		DriveUnit : MC_DriveUnitManager;
		rPositionCleanMotorBwd : REAL; (*Position in mm*)
		rPositionCleanMotorFwd : REAL; (*Position in mm*)
		iMaxSpeedCleanMotorBwd : INT;
		iMaxSpeedCleanMotorFwd : INT;
		iMinSpeedCleanMotorBwd : INT;
		iMinSpeedCleanMotorFwd : INT;
		iCleanMotorSpeedBwd : INT; (*Software Input from a machine value*)
		iCleanMotorSpeedFwd : INT; (*Software Input from a machine value*)
		rMinPrintHeadPos : REAL; (*Minium Print Head Position. Configuration of the machine in mm*)
		rFirstHeadPosition : REAL; (*Software Input. Position of first printhead in mm. Input from a machine value*)
		rLastHeadPosition : REAL; (*Software Input. Position of first printhead in mm. Input from a machine value*)
	END_STRUCT;
	StBlock_Parameters_Motor : 	STRUCT
		DriveUnit : MC_DriveUnitManager;
		rPrintPosition : REAL; (*Input from LC Band. Value in mm*)
		rDriveManSpeed : REAL; (*Vertical motor manual speed. Value in mm/s*)
		rDriveAutoSpeed : REAL; (*Vertical motor automatic speed. Value in mm/s*)
		rCappingPosition : REAL; (*Capped position in mm*)
		rCapPosition : REAL; (*Capped position in mm*)
		rCleanPosition : REAL; (*Clean position in mm*)
		rSafePosition : REAL; (*Position in mm*)
		rMinSafePosition : REAL; (*Position in mm*)
		rWaterSpurtPosition : REAL; (*Position in mm*)
		rSafeMarginForwardTray : REAL; (*Offset para la posicion de seguridad del carro de limpieza. Value in mm*)
		rSafePositionCleanCarrier : REAL; (*Position in mm*)
		rDripBarsPosition : REAL; (*Position in mm*)
		rReferencePosition : REAL; (*Reference Position in mm*)
		rMinThicknessMedia : REAL; (*Minimum media thickness in mm*)
		VerticalDirection : MotorDirection_enum; (*To indicate that the motor must spin in reverse*)
		uiMaxCurrentBarsUp : UINT;
		uiMaxCurrentBarsDown : UINT;
		rReduceSpeedDistance : REAL; (*Distance to the limit to reduce manual speed*)
		rMinCleanOffsetTech : REAL; (*Minimum Cleaning offset by the Technician in mm*)
		rMaxCleanOffsetTech : REAL; (*Maximum Cleaning offset by the Technician in mm*)
		rAcceleration : REAL;
		rDeceleration : REAL;
		xFastSpeedAllowed : BOOL; (*Use of fast speed is allowed*)
		rAutoSpeedMoveUpFast : REAL; (*Bars motor speed to move up fast. Used while in printing to raise position quickly*)
		rAutoSpeedMoveUp : REAL := 50; (*Bars motor speed to move up*)
		rAutoSpeedMoveDown : REAL := 15; (*Bars motor speed to move down*)
		xOversized : BOOL; (*Variable to define motor's operation torque is much lower than the rated torque*)
		rOperationTorque : REAL; (*Motor's operation torque in Nm*)
	END_STRUCT;
	StBlock_SwParameters : 	STRUCT
		xEnableToMovements : BOOL; (*Block is enalbed to movements and doesnt go to print if order is received,  Cleaning? *)
		xEnableToPrint : BOOL; (*Block is enalbed to print and it goes to print if order is received,*)
		rOffsetPrintMotor : REAL; (*Software Input. Printer description, advanced (adjust the motor block position)*)
		rOffsetCleanMtrAdjust : REAL; (*SoftwareInput. Value in mm*)
		rOffsetCleanMtrOperatr : REAL; (*SoftwareInput. Value in mm*)
	END_STRUCT;
	StBlock_Parameters_Hw : 	STRUCT
		xExistBlock : BOOL;
		xThereIsInTraySensor : BOOL;
		xIsWater : BOOL;
		SafetySignals : enumEFI_SafetySignals;
		ValvesNode : USINT;
		ValvesCommsType : CommsNetworkType_enum;
		iNumHeaterPSU : USINT;
		iNumPrintheadsPSU : USINT;
	END_STRUCT;
	StBlock_Parameters : 	STRUCT
		Motor : StBlock_Parameters_Motor;
		Icla : StBlock_Parameters_Icla;
		Inks : StBlock_Parameters_Inks;
		Hw : StBlock_Parameters_Hw;
		tiTimeWaitTrayOutAlarm : TIME; (*Time to position beside headers*)
		tiTimeWaitTrayOut : TIME; (*Time to position beside headers*)
		tiTimeWaitTrayInAlarm : TIME; (*Time to position under headers*)
		tiTimeWaitTrayIn : TIME; (*Time to position under headers*)
		iIclaAxisIndex : USINT; (*Index of the Icla motor to assign it*)
		iMotorAxisIndex : INT; (*Index of the vertical motor to assign it*)
		xPrinterKeyMaintenanceActivated : BOOL; (*Maintenance key activated*)
		xMediaBelow : BOOL; (*The machine send the information that there are media below block*)
		iMappingBlock : INT; (*Defining the physical position of the block. 1= BlockA 2=BlockB*)
		xLeftHandMachine : BOOL; (*To indicate that the machine is left hand.*)
		xRightHandMachine : BOOL; (*To indicate that the machine is right hand.*)
		iFirstBlock : USINT := 1; (*The first block is the number 1 by default*)
		iLastBlock : USINT := 2; (*The second block is the number 2 by default*)
		rManPrintingPos : REAL := 10.0; (*Printing position for manual operation*)
		rPrePrintingPos : REAL; (*Safe printing position in machines with vacuum to protect printheads*)
		iFirstBarPosition : UINT;
		iLastBarPosition : UINT;
		xMotorOffsetAllowed : BOOL; (*Printing position may be modified by using Block.parSw.rOffsetPrintMotor when this variable is activated*)
		xWastedInkTankProcess : BOOL;
		xCappingProcess : BOOL;
		uiCleaningType : USINT; (*0: Undefined  1: Venturi   2: Turbin*)
		iApplicationBars : USINT; (*Number of physical bars that can work for application purposes (inks, curing, ...)*)
	END_STRUCT;
	StBlock_IclaStatus : 	STRUCT
		iIclaState : INT; (*Drive status state machine Icla*)
		xInError : BOOL;
		xHomed : BOOL;
		xIsMoving : BOOL;
		xHoming : BOOL;
		rCurrentPosition : REAL; (*Current position in mm*)
		iSpeed : INT; (*//TODO: Define the units of the speed*)
		iMaxSpeed : INT;
		iIntensityCleanMotor : INT;
		ErrorNumber : UINT;
		rActTemp : REAL; (*Actual temperature*)
		rMaxTemp : REAL;
		rActTorque : REAL;
		rMaxTorque : REAL;
	END_STRUCT;
	StBlock_MotorStatus : 	STRUCT
		xBarsHomed : BOOL;
		xBarsHoming : BOOL;
		ActPosition : UDINT; (*Actual Position of the motor in Motor units*)
		iIntensityVertMotor : INT;
		rMotorAbsPosDesired : REAL;
		rActTemp : REAL; (*Actual temperature*)
		rSpeed : REAL;
		rMaxTemp : REAL;
		iActTorque : INT;
		rRatedTorque : REAL;
		rActTorque : REAL;
		rMaxTorque : REAL;
		rActVelocity : REAL;
		rMaxVelocity : REAL;
		xEnableUp : BOOL;
		xEnableDown : BOOL;
		ErrorID : UINT; (*ErrorID of any occurred error*)
		rOperationTorque : REAL; (*Motor's operation torque*)
	END_STRUCT;
	StBlock_StatusPosition : 	STRUCT
		xUndefined : BOOL;
		xInCap : BOOL;
		xInPrint : BOOL;
		xInClean : BOOL; (*In Clean position. Arrived in Manual*)
		xCleaning : BOOL;
		xGoingToCap : BOOL;
		xGoingToPrint : BOOL;
		xGoingToClean : BOOL;
		xReadyToPrint : BOOL; (*In print postion without safe offsets position*)
	END_STRUCT;
	StBlock_Status : 	STRUCT
		iBlockCaseLogicControl : INT; (*nState logic control*)
		iBlockState : INT; (*Value to send to Sw: 0=NO_AUTO, 1=IN_CAP, 2=IN_PRINT, 3=CLEANING, 4=GOING_TO_CAP, 5=GOING_TO_PRINT*)
		xEnabledMovements : BOOL;
		xAnyManualMovement : BOOL;
		BlockState : Block_States_enum := BLOCK_STOPPING;
		PositionState : Block_Position_enum := BLOCKP_UNDEFINED;
		Position : StBlock_StatusPosition;
		xCleaningDone : BOOL; (*EDGE*)
		xCapOrderDuringCleaning : BOOL;
		xEnabledToPrint : BOOL;
		xEnabledToClean : BOOL;
		xIsWaterBlock : BOOL; (*This Block Is Water*)
		xAlarmToEmptyBelt : BOOL; (*This Block has an alarm that requires to empy the belt*)
		iBarsReadyToPrint : INT;
		rMotorPosition : REAL; (*To Software. Value in mm*)
		execTimes : UDINT;
		Motor : StBlock_MotorStatus;
		Icla : StBlock_IclaStatus;
		ManualCommands : StBlock_Outputs;
		iTemperature : INT; (*Ambient temperature measured (-40..60 ºC)*)
		iHumidity : INT; (*Ambient humidity measured (0..100%)*)
	END_STRUCT;
	StBlock_SafetyInputs : 	STRUCT
		xSafetyOK : BOOL; (*Bar Safety Is Ok*)
		xRearSafetyOK : BOOL; (*Rear Door is OK with Preventa OR LightCourtain is OK in P4*)
		xFrontSafetyOK : BOOL; (*Front Door is Open*)
		xCurtainEnable01 : BOOL;
		xCurtainEnable02 : BOOL;
		xFrontEStopOK : BOOL;
		xRearEStopOK : BOOL;
	END_STRUCT;
	StBlock_Inputs : 	STRUCT
		Safety : StBlock_SafetyInputs;
		xReferenceDI : BOOL;
		xModuleTemp01Ok : BOOL;
		xModuleTemp02Ok : BOOL;
		xModuleTemp03Ok : BOOL;
		xModuleTemp04Ok : BOOL;
		xIclaSensor : BOOL;
		xVertTopLimit : BOOL;
		xTrayIn : BOOL; (*Tray below the bars. Ready to get any drip of the printheads*)
		xTrayOut : BOOL; (*Tray in safe position to move bars to print*)
		xDifferentialOK : BOOL;
		xDriveProtectionOK : BOOL;
		xSiUnitModuleOk : BOOL;
		xIclaModuleOk : BOOL;
		xAirVenturiOK : BOOL;
		xWaterLevelSensor : BOOL; (*Water Tank Minium Level Sensor*)
		xWaterPresureSensor : BOOL; (*Water Presure Sensor*)
		xHeaterDcOkBusBar1 : BOOL; (*Bar Heater Power Supply Work Ok. Signal from a Relay with the coil in the BusBar to confirm voltage*)
		xHeaterDcOkBusBar2 : BOOL; (*Bar Heater Power Supply Work Ok. Signal from a Relay with the coil in the BusBar to confirm voltage*)
		xHeaterDcOkPsu : ARRAY[0..MAX_LAST_HEATER_PSU_DC_OK]OF BOOL; (*Heater Power Supply Work Ok. Signal DC OK from the PSU*)
		xHeaterAcOkPsu : ARRAY[0..MAX_LAST_HEATER_PSU_AC_OK]OF BOOL; (*Heater Power Supply Work Ok. Signal AC  OK from the PSU*)
		xPrintHeadPSU : ARRAY[0..MAX_LAST_PH_PSU]OF BOOL; (*Interconected PrintHead Power Supply Number 1 Work Ok*)
		xCappingWaterLevelSensor : BOOL; (*Sensor checking capping water tank's minimum level*)
		xCappingWaterFlowmeter : BOOL; (*Sensor checking capping water circuit flow*)
		xDegasserPressure : BOOL; (*Pressure switch for degasser pressure control*)
		xFrontDoorClosed : BOOL;
		iTemperatureRaw : INT;
		xTemperatureSensorError : BOOL;
		iHumidityRaw : INT;
		xHumiditySensorError : BOOL;
		xBarsIn : BOOL;
	END_STRUCT;
	StBlock : 	STRUCT
		In : StBlock_Inputs;
		Status : StBlock_Status;
		parameters : StBlock_Parameters;
		parSw : StBlock_SwParameters;
		commands : stBlock_commands; (*all block commands*)
		AlSummary : stEFI_AlarmSummary;
		Al : StBlock_Alarms;
		Lg : StBlock_Log;
		Out : StBlock_Outputs;
	END_STRUCT;
END_TYPE
```

### Block.var
```iecst
VAR
	gIndexBlock : USINT;
END_VAR
```

### Block Docu.txt
```
#################################################################################
#################################################################################
#																				#
#			GENERAL USE OF BLOCK												#
#																				#
# 	To use this BLOCK unit, some general variables are needed:					#
#																				#
# 		gBlock[1..iNumberBlocks] as StBlock										#
#		gAxis[1..iNumberTotalAxis] as AxisCtrl_typ								#
#		gIcla[1..iNumberTotalIclas] as stIcla									#
#		gInks[1..iNumberInks] as stInks.										#
#																				#
#	There are some Libraries needed, too:										#
#		EFILib																	#
#		Libraries (the Global libraries)										#
#																				#
#	And some variables declaration sections:									#
#		GVars: permanent vars are defined in Global.typ., they are needed.		#
#		GStructs: StPermanentGeneral is needed, and it's defined inside it.		#
#																				#
#																				#
#################################################################################
*NOTE: we have maintained Inks as general because we want inks to be an independent functional unit.
So, is for that reason that block needs inks to work. [SEA](06/08/19)

#################################################################################
#################################################################################
#																				#
#			¡¡¡IMPORTANT!!!!													#
# 	Review gAxisCtrl and IclaCtrl for extra needs about 						#
# 	Axis and Icla to use them													#
#																				#
#################################################################################
```

### Program Logical/ExtPack/BlockCtrl/BlockCtrl_v1/BlockCtrl

#### BlockCtrl.var
```iecst
VAR
	iReasonDanger : USINT;
	PositionStateDanger : Block_Position_enum;
	xDangerCollision : BOOL;
	TNotPrinterZero : TON;
	xCleanInterrupt : BOOL;
	reasonSound : UDINT;
	ars_AlrTempPowerSupply : AutoResetSound;
	ars_AlrPHPowerSupply : AutoResetSound;
	ars_AlrAirVenturi : AutoResetSound;
	ars_AlrDif : AutoResetSound;
	ars_AlrCritical : AutoResetSound;
	ars_AlrStop : AutoResetSound;
	ars_AlrWarning : AutoResetSound;
	AxisBK : REFERENCE TO AxisCtrl_typ;
	xMotorHomeOrder : BOOL;
	xFinishedDrippingOrderByBlock : BOOL;
	xIclaAbsMovDone : BOOL; (*Edge*)
	xIclaAbsMovOrder : BOOL; (*State*)
	xCapOrder : BOOL;
	xMotorAbsMovOrder : BOOL; (*Just to Raise the order. It is reseted once sent the information to the Axis*)
	xAnyManualMov : BOOL;
	xStartToCleanOrder : BOOL;
	xOrderToPrint : BOOL;
	xStoppedIclaByTimeActive : BOOL;
	xAnyManualMovement : BOOL;
	xStoppedByExcessiveTimeActive : BOOL;
	xIclaMoving : BOOL;
	rOffseCleanMtr_Copy : REAL;
	rCalcPosDesPrint : REAL; (*Bar's printing position calculation*)
	rMotorAbsPosDesired : REAL; (*Position in mm*)
	rIclaAbsPosDesired : REAL; (*Position desired in mm. pulses 100 pulses per 16mm*)
	rIclaCurrentPos : REAL; (*Position of the Icla in mm*)
	tiDripTimeMax : TIME; (*Maximum Drip time of all the bars of the block*)
	rMotorCurrentPos : REAL; (*Position in mm*)
	iLastState : INT;
	nState : INT := 0;
	iIndexInks : {REDUND_UNREPLICABLE} USINT;
	rOffseCleanMtr : REAL;
	rBlockReductionTempPower : REAL;
	rPowerTempTotalBlock : REAL;
	rsCleaning : RS;
	Block : REFERENCE TO StBlock;
	stBlockCommandsReseted : stBlock_commands;
	stBlockAlarmsReseted : StBlock_Alarms;
	stBlockAlarmsSummaryReseted : stEFI_AlarmSummary;
	IclaBK : REFERENCE TO stIcla;
	T_SafetyError : TOF;
	tonStabInksAfterDrip : TON;
	TON_StoppedIclaByTimeActive : TON;
	TON_excessiveBlockActivated : TON;
	T_IclaError : TON; (*TON Icla error, Error value <> 0*)
	T_DelayAlarmRef : TON;
	T_AlrComsCleanMotor : TON;
	T_AlCleanSensor : TON;
	T_DelayIncoherCleanMtr : TON;
	T_AlrNoPressureWhenWaterPumpIsOn : TON; (*TON top delay water pump alarm when pump is on*)
	TON_AlrTrayOut : TON;
	TON_DRIPPING : TON;
	TON_AlrTrayIn : TON;
	iTimesStopMovWhileHoming : UINT;
	iTimesStateBlockGoingToPrint : USINT;
	iTimesStateBlockCleaning : USINT;
	iTimesStateBlockUndefined : USINT;
	iTimesStateBlockPrinting : USINT;
	iTimesStateBlockGoingToCap : USINT;
	iTimesStateBlockInCap : USINT;
	iTimesStateBlockHomingBar : USINT;
	iTimesStateBlockHomingIcla : USINT;
	xEnableResetIcla : BOOL;
	TON_TrayInSensor : TON;
	MotorDriveUnit : DriveUnitMngr;
	IclaDriveUnit : DriveUnitMngr;
	iReasonStop : UDINT;
	iReasonCritical : UDINT;
	tonWaitingSensor : TON;
	stIclaOrderEventLog : EventLog_typ;
	stIclaEventLog : EventLog_typ;
	VerMotorOrderEventLog : EventLog_typ;
	VerMotorEventLog : EventLog_typ;
	stEventLogCritical : EventLog_typ;
	stEventLogStop : EventLog_typ;
	stEventLogToCap : EventLog_typ;
	stEventLogToPrint : EventLog_typ;
	stEventLogToClean : EventLog_typ;
	stEventLogIncoherence : EventLog_typ;
	stEventLogxHeaterDcOkBusBar1 : EventLog_typ;
	stEventLogxHeaterDcOkBusBar2 : EventLog_typ;
	stEventLogxHeaterDcOkPsu1 : EventLog_typ;
	stEventLogxHeaterDcOkPsu2 : EventLog_typ;
	stEventLogxHeaterDcOkPsu3 : EventLog_typ;
	stEventLogxHeaterAcOkPsu1 : EventLog_typ;
	stEventLogxHeaterAcOkPsu2 : EventLog_typ;
	stEventLogxHeaterAcOkPsu3 : EventLog_typ;
	strAuxEventDesc : STRING[129];
	xChangeMotorSpeedUp : BOOL; (*Signal to change motor speed in manual up movements by near limit*)
	xChangeMotorSpeedDown : BOOL; (*Signal to change motor speed in manual down movements by near limit*)
	TON_DelayAnyVerticalDriveAlarm : TON;
	ars_EmergencyStop : AutoResetSound;
	BlockStatePrevious : Block_States_enum;
	MachineStatePrevious : enumEFI_GenMachineState;
	iCancelHomingBar : UINT;
	BlockPositionPreviousCleaning : Block_Position_enum;
	BlockPositionPrevious : Block_Position_enum;
	iSaveState : UINT;
	iSaveReason : UINT;
	iCancelCleaning : UINT;
	iReasonMovingMan : UINT;
	xAlrToAvoidCleanWithWater : BOOL;
	xBlockPosChange : BOOL;
	xCloseReliefValve : BOOL;
	xInCap : BOOL; (*Internal var to define if the block is in this position*)
	xInPrint : BOOL; (*Internal var to define if the block is in this position*)
	xInClean : BOOL; (*Internal var to define if the block is in this position*)
	rSafeBarPosToCarrier : REAL; (*Position in mm to block Carrier in Manual mode*)
	TOF_CleanOffsetChng : TOF;
	TON_WaitDepresWater : TON; (*TON to wait a few secods to depresre water circuit*)
	TP_WaterSpurtDesactDelay : TP;
	TON_WaitToMoveTrayOut : TON; (*TON to wait a few secods to depresre water circuit*)
	xWaitToMoveTrayOut : BOOL;
	rMoveAboveCapping : REAL := 10.0; (*Distance to move above capping when going to print*)
	TON_AlrCappingWaterNotRecirc : TON; (*TON top delay water pump alarm when pump is on*)
	TP_CappingWaterPumpDesactDelay : TP;
	iReasonAnyWarning : UDINT;
	iReasonSafetyGeneral : UINT;
	iReasonSafetyCutAir : UINT;
	xAnyUpperSafety : BOOL; (*Block.Al.xAlrFrontCurtain OR Block.Al.xAlrRearSafety OR Block.Al.xAlrFrontSafety*)
	tonDelayTraySensorError : TON;
	CanGetState : CANopenGetState;
	tonNotValveComms : TON;
	tonValveCommsErrorResetting : TON;
	ValvesCanResetState : CanOpenResetCommsState_enum;
	ValvesCanResetState_copy : CanOpenResetCommsState_enum;
	CANopenResetValves : CANopenNMT;
	iReasonNotValveComms : UINT;
	xChangedValvesState : BOOL;
	iTimesTryToReset : UINT;
	lastCanOpenResetError : UINT;
	lastResetingState : UINT;
	lastFbResetStatus : UINT;
	ton_TrayOut : TON;
	nStateDanger : UINT;
	ReasonErrorID : UINT;
	ResetManCommands : stBlock_commandsManual;
	ton_ControllerReady : TON;
	xFrontDoorStatusChanged : BOOL;
	xFrontDoorStatus : BOOL;
	xLoggingVerMovingOrder : BOOL;
	TON_OvertorqueWarning : TON;
	tonOvertorqueAlarm : TON;
	Tp_ManWastePump : TP;
	Ton_WastedInkTankPump : TON;
	Ton_CappingPump : TON;
	iIndexHistory : UINT;
	StateGenHistory : ARRAY[0..iHistoryLines] OF Block_States_enum;
	StatePosHistory : ARRAY[0..iHistoryLines] OF Block_Position_enum;
	rMotorAbsPosDesiredPrevious : REAL;
	xStartWastedInkPump : BOOL;
	iReasonRunWastedInkPump : USINT;
	iIndexPsu : USINT;
END_VAR
```
